# B&R Automation Studio project vibratorControlWithCurrentController (part 18)

#### simWing.st
```iecst
ACTION simWing:

	IF wing.activated THEN

		//===============================================================================
		//						Read outputs
		//===============================================================================
		//upperOpen
		wing.hw.out[0].enable := TRUE;
		wing.hw.out[0].pvName := 'upperFlap:this.hw.do_open';
		wing.hw.out[0]();

		//middleOpen
		wing.hw.out[1].enable := TRUE;
		wing.hw.out[1].pvName := 'middleFlap:this.hw.do_open';
		wing.hw.out[1]();

		//bottomOpen
		wing.hw.out[2].enable := TRUE;
		wing.hw.out[2].pvName := 'bottomFlap:this.hw.do_open';
		wing.hw.out[2]();

		//===============================================================================
		//						Set inputs
		//===============================================================================
		//::upperFlap:this.flap.di_changeover
		wing.hw.in[0].enable   := TRUE;
		wing.hw.in[0].dpName   := '%IX.IF6.ST5.DigitalInput01';

		//::middleFlap:this.flap.di_changeover
		wing.hw.in[1].enable   := TRUE;
		wing.hw.in[1].dpName   := '%IX.IF6.ST5.DigitalInput03';

		//::bottomFlap:this.flap.di_changeover
		wing.hw.in[2].enable   := TRUE;
		wing.hw.in[2].dpName   := '%IX.IF6.ST5.DigitalInput02';

		FOR i:=0 TO MAX_WINGS DO
			wing.var.TON_delay[i].PT := T#50ms;
			wing.var.TOF_changeOver[i].PT := T#20ms;
			// check for change
			IF wing.var.oldVal[i] <> wing.hw.out[i].actValue THEN
				wing.var.TON_delay[i].IN := TRUE;
			END_IF
			// after delay time
			wing.var.TOF_changeOver[i].IN := wing.var.TON_delay[i].Q;

			IF wing.var.TOF_changeOver[i].Q THEN
				wing.var.TON_delay[i].IN := FALSE;
				wing.hw.in[i].setValue := 1;
			ELSE
				wing.hw.in[i].setValue := 0;
			END_IF

			wing.var.TON_delay[i]();
			wing.var.TOF_changeOver[i]();
			wing.var.oldVal[i] := wing.hw.out[i].actValue;
		END_FOR

		wing.hw.in[0]();
		wing.hw.in[1]();
		wing.hw.in[2]();

	END_IF

	IF gWingInterface.status.simNeighbour OR wing.activated THEN
		//neighbourBottomOpen
		wing.hw.out[3].enable := TRUE;
		wing.hw.out[3].pvName := 'bottomFlap:this.hw.do_neighbourOpen';
		wing.hw.out[3]();

		//bricksInMiddle
		wing.hw.out[4].enable := TRUE;
		wing.hw.out[4].pvName := 'cassette:this.hw.do_bricksReadyInCassette';
		wing.hw.out[4]();

		//bricksInMiddle
		wing.hw.out[5].enable := TRUE;
		wing.hw.out[5].pvName := 'bottomFlap:this.hw.do_neighbourPortionReady';
		wing.hw.out[5]();

		//::bottomFlap:this.neighbourFlap.di_changeover
		wing.hw.in[3].enable   := TRUE;
		wing.hw.in[3].dpName   := '%IX.IF6.ST5.DigitalInput04';

		 i:=3;
		wing.var.TON_delay[i].PT := T#50ms;
		wing.var.TOF_changeOver[i].PT := T#20ms;
		// check for change
		IF wing.var.oldVal[i] <> wing.hw.out[i].actValue THEN
			wing.var.TON_delay[i].IN := TRUE;
		END_IF
		// after delay time
		wing.var.TOF_changeOver[i].IN := wing.var.TON_delay[i].Q;

		IF wing.var.TOF_changeOver[i].Q THEN
			wing.var.TON_delay[i].IN := FALSE;
			wing.hw.in[i].setValue := 1;
		ELSE
			wing.hw.in[i].setValue := 0;
		END_IF

		wing.var.TON_delay[i]();
		wing.var.TOF_changeOver[i]();
		wing.var.oldVal[i] := wing.hw.out[i].actValue;

		wing.hw.in[3]();

		//::bottomFlap:this.hw.di_neighbourActive
		wing.hw.in[4].enable   := gWingInterface.status.simNeighbour;
		wing.hw.in[4].dpName   := '%IX.IF6.ST6.DigitalInput02';
		wing.hw.in[4].setValue := 1;
		wing.hw.in[4]();

		//::bottomFlap:this.hw.di_neighbourPortionReady
		wing.hw.in[5].enable   :=  gWingInterface.status.simNeighbour;
		wing.hw.in[5].dpName   := '%IX.IF6.ST6.DigitalInput05';
		IF wing.hw.out[5].actValue > 0 THEN
			wing.hw.in[5].setValue := 1;
		ELSE
			wing.hw.in[5].setValue := 0;
		END_IF
		wing.hw.in[5]();

	END_IF

END_ACTION
```

#### simCassette.st
```iecst
ACTION simCassette:

	IF cassette.activated THEN
		gCassetteInterface.cmd.cassetteIsBeingSimulated := TRUE;
		// init sim (TRUE = no box)
		IF EDGEPOS(cassette.activated) THEN
			cassette.hw.in[0].setValue := TRUE;
			cassette.hw.in[1].setValue := TRUE;
		END_IF

		//===============================================================================
		//						Read outputs
		//===============================================================================
		//cassette:this.hw.do_bricksReadyInCassette
		cassette.hw.out[0].enable := TRUE;
		cassette.hw.out[0].pvName := 'cassette:this.hw.do_bricksReadyInCassette';
		cassette.hw.out[0]();

		//cassette:this.hw.do_cassetteRelease
		cassette.hw.out[1].enable := TRUE;
		cassette.hw.out[1].pvName := 'cassette:this.hw.do_cassetteRelease';
		cassette.hw.out[1]();

		//===============================================================================
		//						Set inputs
		//===============================================================================

		cassette.hw.in[0].enable   := TRUE;
		cassette.hw.in[0].dpName   := '%IX.IF6.ST6.DigitalInput03';		//cassette:this.hw.di_cassetteReady

		cassette.hw.in[1].enable   := TRUE;
		cassette.hw.in[1].dpName   := '%IX.IF6.ST6.DigitalInput01';		//cassette:this.hw.di_cassetteQueue

		//cassette:this.hw.di_cassetteQueue
		CASE cassette.var.state OF
			0:
				cassette.hw.in[0].setValue := 0; // no cassette on ready sensor

				cassette.var.tonDelay(IN := TRUE, PT:=cassette.var.toReadyTime);

				IF cassette.var.tonDelay.Q THEN
					cassette.var.tonDelay(IN:=FALSE);
					cassette.var.state := 10;
				END_IF
			10:
				cassette.var.tonDelay(IN := cassette.hw.out[1].actValue > 0, PT:=cassette.var.toReadyTime);

				IF cassette.var.tonDelay.Q THEN
					cassette.var.tonDelay(IN:=FALSE);
					cassette.var.state := 20;
				END_IF

			20:
				cassette.hw.in[0].setValue := 1; // cassette on ready sensor

				cassette.var.tonDelay(IN := TRUE, PT:=cassette.var.fromReadyTime);

				IF cassette.var.tonDelay.Q THEN
					cassette.var.tonDelay(IN:=FALSE);
					cassette.var.tofDelay(IN := TRUE, PT:=cassette.var.cassetteQueueTime);
					cassette.var.state := 0;
				END_IF
		END_CASE

		cassette.var.tofDelay(IN := FALSE, PT:=cassette.var.toReadyTime);
		cassette.hw.in[1].setValue := SEL(cassette.var.tofDelay.Q, 1, 0); // no cassette on queue sensor

	cassette.hw.in[0]();
	cassette.hw.in[1]();

	IF gWingInterface.status.simNeighbour THEN
		//cassette:this.hw.di_neighbourBricksInCassette
		cassette.hw.in[2].enable   := TRUE;
			cassette.hw.in[2].dpName   := '%IX.IF6.ST6.DigitalInput07';
			IF cassette.hw.out[0].actValue > 0 THEN // this machine has brics ready then wing do also.
				cassette.hw.in[2].setValue := 1;
			ELSE
				cassette.hw.in[2].setValue := 0;
			END_IF
		ELSE
			cassette.hw.in[2].enable   := FALSE;
		END_IF
		cassette.hw.in[2]();

	ELSE
		gCassetteInterface.cmd.cassetteIsBeingSimulated := FALSE;
	END_IF

END_ACTION
```

### simGlobal.typ
```iecst
TYPE
	gSimulation_status_typ : 	STRUCT
		photoSensor : BOOL;
		simulateAllButWing : BOOL;
	END_STRUCT;
	gSimulation_typ : 	STRUCT
		status : gSimulation_status_typ;
	END_STRUCT;
END_TYPE
```

### simGlobal.var
```iecst
VAR
	gSimulation : gSimulation_typ;
END_VAR
```

### simCapconGlobal.typ - Global data types
```iecst
TYPE
	gSimCapcon_typ : 	STRUCT
		cmd : gSimCapcon_cmd_typ; (*Command type.*)
		status : gSimCapcon_status_typ; (*Status type.*)
		parameter : gSimCapcon_parameter_typ;
	END_STRUCT;
	gSimCapcon_cmd_typ : 	STRUCT  (*Global command type.*)
		readFile : BOOL;
	END_STRUCT;
	gSimCapcon_status_typ : 	STRUCT  (*Global status type.*)
		data : gSimCapcon_data_typ;
		simSignal : INT;
	END_STRUCT;
	gSimCapcon_parameter_typ : 	STRUCT
		fileName : STRING[200];
	END_STRUCT;
	gSimCapcon_data_typ : 	STRUCT
		record : ARRAY[0..CAPCON_LOG_RECORD_SIZE]OF gSimCapcon_data_record_typ;
	END_STRUCT;
	gSimCapcon_data_record_typ : 	STRUCT
		value : ARRAY[0..CAPCON_LOG_SAMPLE_SIZE]OF INT;
	END_STRUCT;
END_TYPE
```

### simCapconGlobal.var - Global variables
```iecst
VAR
	gSimCapcon : gSimCapcon_typ; (*Global recipe interface.*)
END_VAR
VAR CONSTANT
	CAPCON_LOG_RECORD_SIZE : DINT := 99; (*99 means 100*)
	CAPCON_LOG_SAMPLE_SIZE : DINT := 499; (*499 means 500*)
END_VAR
```

### Program Logical/simulation/capcon/simCapcon (IEC)

#### main.st - Init, cyclic, exit code
```iecst
PROGRAM _INIT

	gSimCapcon.parameter.fileName := 'simData.csv';

	IF gMainInterface.status.simulation THEN
		gSimCapcon.cmd.readFile := TRUE;
	END_IF

END_PROGRAM

PROGRAM _CYCLIC

	CASE cm.state OF

		0:
			cm.description := 'waiting for command';
			IF gSimCapcon.cmd.readFile THEN
				gSimCapcon.cmd.readFile := FALSE;
				cm.state := 100;
			END_IF

		10:

		100:
			cm.description := 'wait for open file ok';
			this.FileOpen_0.enable 	:= TRUE;
			this.FileOpen_0.pDevice := ADR('SIMDATA');
			this.FileOpen_0.pFile 	:= ADR(gSimCapcon.parameter.fileName);
			this.FileOpen_0.mode 	:= fiREAD_ONLY;
			this.FileOpen_0();
			IF this.FileOpen_0.status = ERR_OK THEN
				brdkStrMemSet(ADR(this.tmpData),0,SIZEOF(this.tmpData));
				this.FileRead_0.ident 	:= this.FileOpen_0.ident;
				this.FileRead_0.offset 	:= 0;
				this.FileRead_0.pDest 	:= ADR(this.tmpData);
				this.FileRead_0.len 	:= SIZEOF(this.tmpData);
				this.FileRead_0.enable	:= TRUE;
				cm.state 				:= 110;
			END_IF

		110:
			cm.description := 'waiting for read file';
			this.FileRead_0();
			IF this.FileRead_0.status = ERR_OK THEN
				this.FileRead_0(enable := FALSE);
				this.FileClose_0.enable := TRUE;
				this.FileClose_0.ident 	:= this.FileOpen_0.ident;
				cm.state := 120;
			END_IF

		120:
			cm.description := 'waiting for file close';
			this.FileClose_0();
			IF this.FileClose_0.status = ERR_OK THEN
				this.FileOpen_0(enable := FALSE);
				this.FileClose_0(enable := FALSE);
				this.lfCnt := 0;
				this.offset := 0;
				brdkStrMemSet(ADR(this.tmpStr),0,SIZEOF(this.tmpStr));
				cm.state := 130;
			END_IF

		130:
			cm.description := 'parse a line';
			FOR this.offset := this.offset TO MAX_FILE_SIZE DO
				CASE this.tmpData[this.offset] OF

					0:	// found end of file
						cm.state := 0;
						EXIT;

					10: // found a line feed
						this.lfCnt 		:= this.lfCnt + 1;
						this.colCnt 	:= 0;					// reset ; count

					59:	// found a ;
						IF this.lfCnt >= START_LINE_FEEDS AND this.colCnt >= START_COLS AND this.colCnt <= MAX_COLS THEN
							gSimCapcon.status.data.record[this.lfCnt - START_LINE_FEEDS].value[this.colCnt - START_COLS] := DINT_TO_INT(brdkStrAToDint(ADR(this.tmpStr),BRDK_STR_CONVERT_DECIMAL));
							brdkStrMemSet(ADR(this.tmpStr),0,SIZEOF(this.tmpStr));
							this.charCnt := 0;
						END_IF
						this.colCnt := this.colCnt + 1;

					32..57:	// numbers and some signs
						IF this.lfCnt >= START_LINE_FEEDS AND this.colCnt >= START_COLS AND this.colCnt <= MAX_COLS THEN
							this.tmpStr[this.charCnt] := this.tmpData[this.offset];
							this.charCnt := this.charCnt + 1;
						END_IF

				END_CASE

			END_FOR

	END_CASE

	cm;

END_PROGRAM

PROGRAM _EXIT
	(* Insert code here *)

END_PROGRAM
```

#### types.typ - Local data types
```iecst
TYPE
	local_typ : 	STRUCT
		FileOpen_0 : FileOpen;
		FileRead_0 : FileRead;
		FileClose_0 : FileClose;
		tmpData : ARRAY[0..MAX_FILE_SIZE]OF USINT;
		offset : UDINT;
		tmpStr : ARRAY[0..9]OF USINT;
		colCnt : UINT;
		lfCnt : USINT;
		charCnt : USINT;
	END_STRUCT;
END_TYPE
```

#### variables.var - Local variables
```iecst
VAR
	this : local_typ;
END_VAR
VAR CONSTANT
	MAX_FILE_SIZE : UDINT := 1000000;
END_VAR
VAR
	cm : brdkCM;
END_VAR
VAR CONSTANT
	MAX_COLS : UINT := 499; (*maximum number of ;*)
	START_COLS : UINT := 2; (*number of ; in a line before the data is good*)
	START_LINE_FEEDS : USINT := 5; (*number of line feeds before the data is good*)
END_VAR
```

### Data object Logical/gAxisVibCobj/gAxisVibCi (Ax)

#### gAxisVibCi.ax
```
InitParameter (Version=5.23.1, NcSwId=ACP10)
  ACP10AXIS_typ:
    dig_in:
      level:
        reference = ncACTIV_HI
        pos_hw_end = ncACTIV_HI
        neg_hw_end = ncACTIV_HI
        trigger1 = ncACTIV_HI
        trigger2 = ncACTIV_HI
    encoder_if:
      parameter:
        count_dir = ncSTANDARD
        scaling:
          load:
            units = 1000
            rev_motor = 1
    limit:
      parameter:
        v_pos = 54000.0
        v_neg = 54000.0
        a1_pos = 5000000.0
        a2_pos = 5000000.0
        a1_neg = 5000000.0
        a2_neg = 5000000.0
        t_jolt = 0.0
        t_in_pos = 0.0
        pos_sw_end = 8388607
        neg_sw_end = -8388608
        ds_warning = 500.0
        ds_stop = 1000.0
        a_stop = 1.0E+30
        dv_stop = 0.0
        dv_stop_mode = ncOFF
    controller:
      mode = ncUF
      position:
        kv = 50.0
        tn = 0.0
        t_predict = 0.0004
        t_total = 0.0004
        p_max = 1.0E+30
        i_max = 0.0
      speed:
        kv = 2.0
        tn = 0.0
        t_filter = 0.0
        isq_filter1:
          type = ncOFF
          a0 = 0.0
          a1 = 0.0
          b0 = 0.0
          b1 = 0.0
          b2 = 0.0
          c0_par_id = 0
          c1_par_id = 0
        isq_filter2:
          type = ncOFF
          a0 = 0.0
          a1 = 0.0
          b0 = 0.0
          b1 = 0.0
          b2 = 0.0
          c0_par_id = 0
          c1_par_id = 0
        isq_filter3:
          type = ncOFF
          a0 = 0.0
          a1 = 0.0
          b0 = 0.0
          b1 = 0.0
          b2 = 0.0
          c0_par_id = 0
          c1_par_id = 0
      uf:
        type = ncLINEAR
        auto_config = ncOFF
        u0 = 0.0
        un = 0.0
        fn = 50.0
        k_f_slip = 0.0
      ff:
        mode = ncSTANDARD
        torque_load = 0.0
        torque_pos = 0.0
        torque_neg = 0.0
        kv_torque = 0.0
        inertia = 0.0
        t_filter_a = 0.0
      fb:
        mode = ncSTANDARD
        speed_mix_ratio = 0.0
        speed_kv = 2.0
      model:
        mass1:
          inertia = 0.0
          viscous_friction = 0.0
        mass2:
          inertia = 0.0
          viscous_friction = 0.0
          stiffness = 0.0
          damping = 0.0
    move:
      stop:
        parameter[0]:
          decel_ramp = ncA_LIMIT
          controller = ncON
        parameter[1]:
          decel_ramp = ncA_LIMIT
          controller = ncON
        parameter[2]:
          decel_ramp = ncA_LIMIT
          controller = ncON
        parameter[3]:
          decel_ramp = ncA_LIMIT
          controller = ncON
        quickstop:
          decel_ramp = ncA_LIMIT
          t_jolt = 0.0
        drive_error:
          decel_ramp = ncA_LIMIT
      homing:
        parameter:
          s = 0
          v_switch = 5000.0
          v_trigger = 500.0
          a = 50000.0
          mode = ncDIRECT
          edge_sw = ncPOSITIVE
          start_dir = ncPOSITIVE
          trigg_dir = ncPOSITIVE
          ref_pulse = ncOFF
          fix_dir = ncOFF
          tr_s_block = 0.0
          torque_lim = 0.0
          ds_block = 0.0
          ds_stop = 0.0
      basis:
        parameter:
          v_pos = 50000.0
          v_neg = 50000.0
          a1_pos = 500000.0
          a2_pos = 500000.0
          a1_neg = 500000.0
          a2_neg = 500000.0
    message:
      text:
        parameter:
          format = ncZERO
          columns = 81
          data_modul = acp10etxen
```

### Data object Logical/gAxisVibCobj/cfCurCtr (Apt)

#### cfCurCtr.apt
```
AcoposParameterTable:
  Root Parameters:
    128 = 1 (Name=SGEN_SW_END_IGNORE)  // Limit values: Ignore SW end positions
    652 = 0 (Name=MOTOR_ENCOD_ATTR)  // Motor: Encoder: Attribute
    1215 = 0 (Name=MOTOR_TEMPSENS_TYPE)  // Temperature sensor: Type
    90 = 76 (Name=BRAKE_MODE)  // Motor holding brake: Mode
    1208 = 1 (Name=MOTOR_NUM_PHASES)  // Motor: Number of motor phases
    Axis Parameter Identification, Synchronous Motor:
      Group  // General Parameters
        30 = 2 (Name=MOTOR_TYPE)  // Motor: Type
        31 = 0x0203 (Name=MOTOR_COMPATIBILITY)  // Motor: Software compatibility
        46 = 1 (Name=MOTOR_WIND_CONNECT)  // Motor: Winding connection
        62 = 0 (Name=MOTOR_INERTIA, Unit=kgm²)  // Motor: Moment of inertia
        849 = 0 (Name=MOTOR_TAU_THERM, Unit=s)  // Motor: Thermal time constant
      Group  // Brake Parameters
        42 = 0 (Name=MOTOR_BRAKE_CURR_RATED, Unit=A)  // Motor holding brake: Rated current
        43 = 0 (Name=MOTOR_BRAKE_TORQ_RATED, Unit=Nm)  // Motor holding brake: Rated torque
        44 = 0 (Name=MOTOR_BRAKE_ON_TIME, Unit=s)  // Motor holding brake: Engaging delay
        45 = 0 (Name=MOTOR_BRAKE_OFF_TIME, Unit=s)  // Motor holding brake: Release delay
      Group  // Thermo Sensor Parameters
        64 = 0 (Name=MOTOR_TEMPSENS_PAR1)  // Temperature sensor: Parameter 1
        65 = 0 (Name=MOTOR_TEMPSENS_PAR2)  // Temperature sensor: Parameter 2
        66 = 0 (Name=MOTOR_TEMPSENS_PAR3)  // Temperature sensor: Parameter 3
        67 = 0 (Name=MOTOR_TEMPSENS_PAR4)  // Temperature sensor: Parameter 4
        68 = 0 (Name=MOTOR_TEMPSENS_PAR5)  // Temperature sensor: Parameter 5
        69 = 0 (Name=MOTOR_TEMPSENS_PAR6)  // Temperature sensor: Parameter 6
        70 = 0 (Name=MOTOR_TEMPSENS_PAR7)  // Temperature sensor: Parameter 7
        71 = 0 (Name=MOTOR_TEMPSENS_PAR8)  // Temperature sensor: Parameter 8
        72 = 0 (Name=MOTOR_TEMPSENS_PAR9)  // Temperature sensor: Parameter 9
        73 = 0 (Name=MOTOR_TEMPSENS_PAR10)  // Temperature sensor: Parameter 10
        74 = 50 (Name=MOTOR_WIND_TEMP_MAX, Unit=°C)  // Temperature sensor: Limit temperature
      Group  // Result Parameters of Parameter Identification
        47 = 1 (Name=MOTOR_POLEPAIRS)  // Motor: Number of pole-pairs
        48 = 200 (Name=MOTOR_VOLTAGE_RATED, Unit=V)  // Motor: Rated voltage
        50 = 6000 (Name=MOTOR_SPEED_RATED, Unit=1/min)  // Motor: Rated speed
        51 = 6600 (Name=MOTOR_SPEED_MAX, Unit=1/min)  // Motor: Maximum speed
        52 = 1 (Name=MOTOR_TORQ_STALL, Unit=Nm)  // Motor: Stall torque
        53 = 1 (Name=MOTOR_TORQ_RATED, Unit=Nm)  // Motor: Rated torque
        54 = 1 (Name=MOTOR_TORQ_MAX, Unit=Nm)  // Motor: Peak torque
        56 = 1 (Name=MOTOR_CURR_STALL, Unit=A)  // Motor: Stall current
        58 = 4 (Name=MOTOR_CURR_MAX, Unit=A)  // Motor: Peak current
        57 = 3.77 (Name=MOTOR_CURR_RATED, Unit=A)  // Motor: Rated current
        59 = 1 (Name=MOTOR_WIND_CROSS_SECT, Unit=mm²)  // Motor: Line cross section
        60 = 6.917 (Name=MOTOR_STATOR_RESISTANCE, Unit=Ohm)  // Motor: Stator resistance
        61 = 0.3237 (Name=MOTOR_STATOR_INDUCTANCE, Unit=Henry)  // Motor: Stator inductance
        1208 = 1 (Name=MOTOR_NUM_PHASES)  // Motor: Number of motor phases
      IPL:
        777 = IPL_MODE+0 (Name=FUNCTION_BLOCK_CREATE, Disabled=FALSE)  // Function block: Create a FB instance
        8712 = USER_R4_VAR1 (Name=IPL_IN_PARID+0, Disabled=FALSE)  // FB0 FB IPL: Parameter ID of input
        8760 = CYCLIC_TODRV_COUNT (Name=IPL_EV_PARID+0)  // FB0 FB IPL: Parameter ID of event input
        8720 = 800 (Name=IPL_CYCLE_TIME+0, Unit=us)  // FB0 FB IPL: Cycle time
        8704 = 2 (Name=IPL_MODE+0, Disabled=FALSE)  // FB0 FB IPL: Mode - (4) quadric no overshoot
      Group:
        347 = 10000 (Name=F_SWITCH, Unit=cps)  // Inverter: Switch frequency
        49 = 100 (Name=MOTOR_VOLTAGE_CONST, Unit=mV*min)  // Motor: Voltage constant
        813 = 0  // PARID_SIGEN_OFFS
        55 = 3 (Name=MOTOR_TORQ_CONST, Unit=Nm/A)  // Motor: Torque constant
        63 = 0 (Name=MOTOR_COMMUT_OFFSET, Unit=rad)  // Motor: Commutation offset
        713 = 8752 (Name=ICTRL_SET_PARID)  // CTRL Current controller: Set value parameter ID of stator current quadrature component
        1480 = 0 (Name=TLIM_MODE)  // CTRL Torque limiter: Mode
        1569 = 2500 (Name=ICTRL_US_FILTER1_A0)  // CTRL Current: Set voltage filter coefficient A0
        1570 = 2200 (Name=ICTRL_US_FILTER1_A1)  // CTRL Current: Set voltage filter coefficient A1
        1568 = 1 (Name=ICTRL_US_FILTER_TYPE)  // CTRL Current: Set voltage filter type
        1166 = 0 (Name=ICTRL_AUTO_CONFIG)  // CTRL Current: Automatic configuration
        223 = 300 (Name=ICTRL_KV, Unit=V/A)  // CTRL Current controller: Proportional amplification factor
        225 = 0.00526 (Name=ICTRL_TI, Unit=s)  // CTRL Current controller: Integral action time
        328 = 5 (Name=CONTROLLER_MODE)  // CTRL Controller: Mode
      Voltage observer:
        1354 = 1 (Name=OBS_MODE_BITS)  // Observer: Mode bits
        1298 = 25.4481 (Name=OBS_VOLT_INVCL_A1)  // Voltage observer: Inverter adjustment amplification factor
        1299 = 2.2113 (Name=OBS_VOLT_INVCL_A2, Unit=1/A)  // Voltage observer: Inverter adjustment exponent
    232 = 0 (Name=CYCLIC_TODRV_PAR_INDEX)  // Cyclic communication: Parameter index of data to drive
    207 = CYCLIC_FRDRV_REC_INDEX (Name=CYCLIC_TODRV_PARID)  // Cyclic communication: Parameter ID of data to drive
    777 = ARITH_MODE+0 (Name=FUNCTION_BLOCK_CREATE)  // Function block: Create a FB instance
    777 = DYNSYS_MODE+0 (Name=FUNCTION_BLOCK_CREATE)  // Function block: Create a FB instance
    777 = ARITH_MODE+1 (Name=FUNCTION_BLOCK_CREATE)  // Function block: Create a FB instance
    777 = ARITH_MODE+2 (Name=FUNCTION_BLOCK_CREATE)  // Function block: Create a FB instance
    777 = DYNSYS_MODE+1 (Name=FUNCTION_BLOCK_CREATE)  // Function block: Create a FB instance
    777 = DYNSYS_MODE+2 (Name=FUNCTION_BLOCK_CREATE)  // Function block: Create a FB instance
    777 = DYNSYS_MODE+3 (Name=FUNCTION_BLOCK_CREATE)  // Function block: Create a FB instance
    777 = DYNSYS_MODE+4 (Name=FUNCTION_BLOCK_CREATE)  // Function block: Create a FB instance
    777 = VAR_I4_0+0 (Name=FUNCTION_BLOCK_CREATE)  // Function block: Create a FB instance
    777 = VAR_R4_0+0 (Name=FUNCTION_BLOCK_CREATE)  // Function block: Create a FB instance
    777 = MINMAX_MODE+0 (Name=FUNCTION_BLOCK_CREATE)  // Function block: Create a FB instance
    777 = MINMAX_MODE+1 (Name=FUNCTION_BLOCK_CREATE)  // Function block: Create a FB instance
    777 = COUNT_MODE+0 (Name=FUNCTION_BLOCK_CREATE)  // Function block: Create a FB instance
    777 = FILTER_MODE+0 (Name=FUNCTION_BLOCK_CREATE)  // Function block: Create a FB instance
    ARITH EMF:
      3584 = 0 (Name=ARITH_MODE+0)  // FB0 ARITH Mode
      3592 = 216 (Name=ARITH_IN1_PARID+0)  // FB0 ARITH Parameter ID of input1
      3600 = 214 (Name=ARITH_IN2_PARID+0)  // FB0 ARITH Parameter ID of input2
      3632 = 1 (Name=ARITH_K1+0)  // FB0 ARITH Multiplication factor1
      3640 = -4.2 (Name=ARITH_K2+0)  // FB0 ARITH Multiplication factor2
      3584 = 4 (Name=ARITH_MODE+0)  // FB0 ARITH Mode
    DYNSYS Integrate EMF:
      14336 = 0 (Name=DYNSYS_MODE+0)  // FB0 FB DYNSYS: Mode
      14344 = 0.99 (Name=DYNSYS_PAR_A+0)  // FB0 FB DYNSYS: System parameter A
      14344 = 0.0002 (Name=DYNSYS_PAR_A+0)  // FB0 FB DYNSYS: System parameter A
      14344 = 0 (Name=DYNSYS_PAR_A+0)  // FB0 FB DYNSYS: System parameter A
      14344 = 0 (Name=DYNSYS_PAR_A+0)  // FB0 FB DYNSYS: System parameter A
      14344 = 0 (Name=DYNSYS_PAR_A+0)  // FB0 FB DYNSYS: System parameter A
      14344 = 0 (Name=DYNSYS_PAR_A+0)  // FB0 FB DYNSYS: System parameter A
      14344 = 0 (Name=DYNSYS_PAR_A+0)  // FB0 FB DYNSYS: System parameter A
      14344 = 0 (Name=DYNSYS_PAR_A+0)  // FB0 FB DYNSYS: System parameter A
      14344 = 0 (Name=DYNSYS_PAR_A+0)  // FB0 FB DYNSYS: System parameter A
      14352 = 0.0002 (Name=DYNSYS_PAR_B+0)  // FB0 FB DYNSYS: System parameter B
      14352 = 0 (Name=DYNSYS_PAR_B+0)  // FB0 FB DYNSYS: System parameter B
      14352 = 1 (Name=DYNSYS_PAR_B+0)  // FB0 FB DYNSYS: System parameter B
      14352 = 0 (Name=DYNSYS_PAR_B+0)  // FB0 FB DYNSYS: System parameter B
      14352 = 0 (Name=DYNSYS_PAR_B+0)  // FB0 FB DYNSYS: System parameter B
      14352 = 1 (Name=DYNSYS_PAR_B+0)  // FB0 FB DYNSYS: System parameter B
      14360 = 1 (Name=DYNSYS_PAR_C+0)  // FB0 FB DYNSYS: System parameter C
      14360 = 0 (Name=DYNSYS_PAR_C+0)  // FB0 FB DYNSYS: System parameter C
      14360 = 0 (Name=DYNSYS_PAR_C+0)  // FB0 FB DYNSYS: System parameter C
      14360 = 0 (Name=DYNSYS_PAR_C+0)  // FB0 FB DYNSYS: System parameter C
      14360 = 0 (Name=DYNSYS_PAR_C+0)  // FB0 FB DYNSYS: System parameter C
      14360 = 1 (Name=DYNSYS_PAR_C+0)  // FB0 FB DYNSYS: System parameter C
      14408 = ARITH_VALUE_R4+0 (Name=DYNSYS_IN1_PARID+0)  // FB0 FB DYNSYS: Parameter ID for input 1
      14416 = 214 (Name=DYNSYS_IN2_PARID+0)  // FB0 FB DYNSYS: Parameter ID for input 2
      14336 = 1 (Name=DYNSYS_MODE+0)  // FB0 FB DYNSYS: Mode (note: set SCTRL_ADD_SET_PARID = DYNSYS_OUT1_VALUE+X for activation)
    ARITH Airgap:
      3585 = 0 (Name=ARITH_MODE+1)  // FB0 ARITH Mode
      3593 = DYNSYS_OUT2_VALUE+0 (Name=ARITH_IN1_PARID+1)  // FB0 ARITH Parameter ID of input1
      3601 = DYNSYS_OUT1_VALUE+0 (Name=ARITH_IN2_PARID+1)  // FB0 ARITH Parameter ID of input2
      3585 = 5 (Name=ARITH_MODE+1)  // FB0 ARITH Mode
    ARITH Observer:
      3586 = 0 (Name=ARITH_MODE+2)  // FB2 FB ARITH: Mode
      3594 = 1296 (Name=ARITH_IN1_PARID+2)  // FB2 FB ARITH: Parameter ID of input1
      3602 = 1297 (Name=ARITH_IN2_PARID+2)  // FB2 FB ARITH: Parameter ID of input2
      3586 = 2 (Name=ARITH_MODE+2)  // FB2 FB ARITH: Mode
    DYNSYS+1:
      14337 = 0 (Name=DYNSYS_MODE+1)  // FB0 FB DYNSYS: Mode
      14345 = 0 (Name=DYNSYS_PAR_A+1)  // FB0 FB DYNSYS: System parameter A
      14345 = 0 (Name=DYNSYS_PAR_A+1)  // FB0 FB DYNSYS: System parameter A
      14345 = 0 (Name=DYNSYS_PAR_A+1)  // FB0 FB DYNSYS: System parameter A
      14345 = 0 (Name=DYNSYS_PAR_A+1)  // FB0 FB DYNSYS: System parameter A
      14345 = 1 (Name=DYNSYS_PAR_A+1)  // FB0 FB DYNSYS: System parameter A
      14345 = 0 (Name=DYNSYS_PAR_A+1)  // FB0 FB DYNSYS: System parameter A
      14345 = 0 (Name=DYNSYS_PAR_A+1)  // FB0 FB DYNSYS: System parameter A
      14345 = 0 (Name=DYNSYS_PAR_A+1)  // FB0 FB DYNSYS: System parameter A
      14345 = 0 (Name=DYNSYS_PAR_A+1)  // FB0 FB DYNSYS: System parameter A
      14345 = 1 (Name=DYNSYS_PAR_A+1)  // FB0 FB DYNSYS: System parameter A
      14345 = 0 (Name=DYNSYS_PAR_A+1)  // FB0 FB DYNSYS: System parameter A
      14345 = 0 (Name=DYNSYS_PAR_A+1)  // FB0 FB DYNSYS: System parameter A
      14345 = 0 (Name=DYNSYS_PAR_A+1)  // FB0 FB DYNSYS: System parameter A
      14345 = 0 (Name=DYNSYS_PAR_A+1)  // FB0 FB DYNSYS: System parameter A
      14345 = 1 (Name=DYNSYS_PAR_A+1)  // FB0 FB DYNSYS: System parameter A
      14345 = 0 (Name=DYNSYS_PAR_A+1)  // FB0 FB DYNSYS: System parameter A
      14353 = 1 (Name=DYNSYS_PAR_B+1)  // FB1 FB DYNSYS: System parameter B
      14353 = 0 (Name=DYNSYS_PAR_B+1)  // FB1 FB DYNSYS: System parameter B
      14353 = 0 (Name=DYNSYS_PAR_B+1)  // FB1 FB DYNSYS: System parameter B
      14353 = 0 (Name=DYNSYS_PAR_B+1)  // FB1 FB DYNSYS: System parameter B
      14361 = 1 (Name=DYNSYS_PAR_C+1)  // FB1 FB DYNSYS: System parameter C
      14361 = 0 (Name=DYNSYS_PAR_C+1)  // FB1 FB DYNSYS: System parameter C
      14361 = 0 (Name=DYNSYS_PAR_C+1)  // FB1 FB DYNSYS: System parameter C
      14361 = 0 (Name=DYNSYS_PAR_C+1)  // FB1 FB DYNSYS: System parameter C
      14361 = 0 (Name=DYNSYS_PAR_C+1)  // FB1 FB DYNSYS: System parameter C
      14361 = 1 (Name=DYNSYS_PAR_C+1)  // FB1 FB DYNSYS: System parameter C
      14361 = 0 (Name=DYNSYS_PAR_C+1)  // FB1 FB DYNSYS: System parameter C
      14361 = 0 (Name=DYNSYS_PAR_C+1)  // FB1 FB DYNSYS: System parameter C
      14409 = 216 (Name=DYNSYS_IN1_PARID+1)  // FB0 FB DYNSYS: Parameter ID for input 1
      14337 = 1 (Name=DYNSYS_MODE+1)  // FB0 FB DYNSYS: Mode (note: set SCTRL_ADD_SET_PARID = DYNSYS_OUT1_VALUE+X for activation)
    DYNSYS+2:
      14338 = 0 (Name=DYNSYS_MODE+2)  // FB0 FB DYNSYS: Mode
      14346 = 0 (Name=DYNSYS_PAR_A+2)  // FB0 FB DYNSYS: System parameter A
      14346 = 0 (Name=DYNSYS_PAR_A+2)  // FB0 FB DYNSYS: System parameter A
      14346 = 0 (Name=DYNSYS_PAR_A+2)  // FB0 FB DYNSYS: System parameter A
      14346 = 0 (Name=DYNSYS_PAR_A+2)  // FB0 FB DYNSYS: System parameter A
      14346 = 1 (Name=DYNSYS_PAR_A+2)  // FB0 FB DYNSYS: System parameter A
      14346 = 0 (Name=DYNSYS_PAR_A+2)  // FB0 FB DYNSYS: System parameter A
      14346 = 0 (Name=DYNSYS_PAR_A+2)  // FB0 FB DYNSYS: System parameter A
      14346 = 0 (Name=DYNSYS_PAR_A+2)  // FB0 FB DYNSYS: System parameter A
      14346 = 0 (Name=DYNSYS_PAR_A+2)  // FB0 FB DYNSYS: System parameter A
      14346 = 1 (Name=DYNSYS_PAR_A+2)  // FB0 FB DYNSYS: System parameter A
      14346 = 0 (Name=DYNSYS_PAR_A+2)  // FB0 FB DYNSYS: System parameter A
      14346 = 0 (Name=DYNSYS_PAR_A+2)  // FB0 FB DYNSYS: System parameter A
      14346 = 0 (Name=DYNSYS_PAR_A+2)  // FB0 FB DYNSYS: System parameter A
      14346 = 0 (Name=DYNSYS_PAR_A+2)  // FB0 FB DYNSYS: System parameter A
      14346 = 1 (Name=DYNSYS_PAR_A+2)  // FB0 FB DYNSYS: System parameter A
      14346 = 0 (Name=DYNSYS_PAR_A+2)  // FB0 FB DYNSYS: System parameter A
      14354 = 1 (Name=DYNSYS_PAR_B+2)  // FB2 FB DYNSYS: System parameter B
      14354 = 0 (Name=DYNSYS_PAR_B+2)  // FB2 FB DYNSYS: System parameter B
      14354 = 0 (Name=DYNSYS_PAR_B+2)  // FB2 FB DYNSYS: System parameter B
      14354 = 0 (Name=DYNSYS_PAR_B+2)  // FB2 FB DYNSYS: System parameter B
      14362 = 0 (Name=DYNSYS_PAR_C+2)  // FB2 FB DYNSYS: System parameter C
      14362 = 0 (Name=DYNSYS_PAR_C+2)  // FB2 FB DYNSYS: System parameter C
      14362 = 1 (Name=DYNSYS_PAR_C+2)  // FB2 FB DYNSYS: System parameter C
      14362 = 0 (Name=DYNSYS_PAR_C+2)  // FB2 FB DYNSYS: System parameter C
      14362 = 0 (Name=DYNSYS_PAR_C+2)  // FB2 FB DYNSYS: System parameter C
      14362 = 0 (Name=DYNSYS_PAR_C+2)  // FB2 FB DYNSYS: System parameter C
      14362 = 0 (Name=DYNSYS_PAR_C+2)  // FB2 FB DYNSYS: System parameter C
      14362 = 1 (Name=DYNSYS_PAR_C+2)  // FB2 FB DYNSYS: System parameter C
      14410 = 216 (Name=DYNSYS_IN1_PARID+2)  // FB0 FB DYNSYS: Parameter ID for input 1
      14338 = 1 (Name=DYNSYS_MODE+2)  // FB0 FB DYNSYS: Mode (note: set SCTRL_ADD_SET_PARID = DYNSYS_OUT1_VALUE+X for activation)
    DYNSYS+3:
      14339 = 0 (Name=DYNSYS_MODE+3)  // FB3 FB DYNSYS: Mode
      14347 = 0 (Name=DYNSYS_PAR_A+3)  // FB3 FB DYNSYS: System parameter A
      14347 = 0 (Name=DYNSYS_PAR_A+3)  // FB3 FB DYNSYS: System parameter A
      14347 = 0 (Name=DYNSYS_PAR_A+3)  // FB3 FB DYNSYS: System parameter A
      14347 = 0 (Name=DYNSYS_PAR_A+3)  // FB3 FB DYNSYS: System parameter A
      14347 = 1 (Name=DYNSYS_PAR_A+3)  // FB3 FB DYNSYS: System parameter A
      14347 = 0 (Name=DYNSYS_PAR_A+3)  // FB3 FB DYNSYS: System parameter A
      14347 = 0 (Name=DYNSYS_PAR_A+3)  // FB3 FB DYNSYS: System parameter A
      14347 = 0 (Name=DYNSYS_PAR_A+3)  // FB3 FB DYNSYS: System parameter A
      14347 = 0 (Name=DYNSYS_PAR_A+3)  // FB3 FB DYNSYS: System parameter A
      14347 = 1 (Name=DYNSYS_PAR_A+3)  // FB3 FB DYNSYS: System parameter A
      14347 = 0 (Name=DYNSYS_PAR_A+3)  // FB3 FB DYNSYS: System parameter A
      14347 = 0 (Name=DYNSYS_PAR_A+3)  // FB3 FB DYNSYS: System parameter A
      14347 = 0 (Name=DYNSYS_PAR_A+3)  // FB3 FB DYNSYS: System parameter A
      14347 = 0 (Name=DYNSYS_PAR_A+3)  // FB3 FB DYNSYS: System parameter A
      14347 = 1 (Name=DYNSYS_PAR_A+3)  // FB3 FB DYNSYS: System parameter A
      14347 = 0 (Name=DYNSYS_PAR_A+3)  // FB3 FB DYNSYS: System parameter A
      14355 = 1 (Name=DYNSYS_PAR_B+3)  // FB3 FB DYNSYS: System parameter B
      14355 = 0 (Name=DYNSYS_PAR_B+3)  // FB3 FB DYNSYS: System parameter B
      14355 = 0 (Name=DYNSYS_PAR_B+3)  // FB3 FB DYNSYS: System parameter B
      14355 = 0 (Name=DYNSYS_PAR_B+3)  // FB3 FB DYNSYS: System parameter B
      14363 = 1 (Name=DYNSYS_PAR_C+3)  // FB3 FB DYNSYS: System parameter C
      14363 = 0 (Name=DYNSYS_PAR_C+3)  // FB3 FB DYNSYS: System parameter C
      14363 = 0 (Name=DYNSYS_PAR_C+3)  // FB3 FB DYNSYS: System parameter C
      14363 = 0 (Name=DYNSYS_PAR_C+3)  // FB3 FB DYNSYS: System parameter C
      14363 = 0 (Name=DYNSYS_PAR_C+3)  // FB3 FB DYNSYS: System parameter C
      14363 = 1 (Name=DYNSYS_PAR_C+3)  // FB3 FB DYNSYS: System parameter C
      14363 = 0 (Name=DYNSYS_PAR_C+3)  // FB3 FB DYNSYS: System parameter C
      14363 = 0 (Name=DYNSYS_PAR_C+3)  // FB3 FB DYNSYS: System parameter C
      14411 = 214 (Name=DYNSYS_IN1_PARID+3)  // FB3 FB DYNSYS: Parameter ID for input 1
      14339 = 1 (Name=DYNSYS_MODE+3)  // FB3 FB DYNSYS: Mode
    DYNSYS+4:
      14340 = 0 (Name=DYNSYS_MODE+4)  // FB4 FB DYNSYS: Mode
      14348 = 0 (Name=DYNSYS_PAR_A+4)  // FB4 FB DYNSYS: System parameter A
      14348 = 0 (Name=DYNSYS_PAR_A+4)  // FB4 FB DYNSYS: System parameter A
      14348 = 0 (Name=DYNSYS_PAR_A+4)  // FB4 FB DYNSYS: System parameter A
      14348 = 0 (Name=DYNSYS_PAR_A+4)  // FB4 FB DYNSYS: System parameter A
      14348 = 1 (Name=DYNSYS_PAR_A+4)  // FB4 FB DYNSYS: System parameter A
      14348 = 0 (Name=DYNSYS_PAR_A+4)  // FB4 FB DYNSYS: System parameter A
      14348 = 0 (Name=DYNSYS_PAR_A+4)  // FB4 FB DYNSYS: System parameter A
      14348 = 0 (Name=DYNSYS_PAR_A+4)  // FB4 FB DYNSYS: System parameter A
      14348 = 0 (Name=DYNSYS_PAR_A+4)  // FB4 FB DYNSYS: System parameter A
      14348 = 1 (Name=DYNSYS_PAR_A+4)  // FB4 FB DYNSYS: System parameter A
      14348 = 0 (Name=DYNSYS_PAR_A+4)  // FB4 FB DYNSYS: System parameter A
      14348 = 0 (Name=DYNSYS_PAR_A+4)  // FB4 FB DYNSYS: System parameter A
      14348 = 0 (Name=DYNSYS_PAR_A+4)  // FB4 FB DYNSYS: System parameter A
      14348 = 0 (Name=DYNSYS_PAR_A+4)  // FB4 FB DYNSYS: System parameter A
      14348 = 1 (Name=DYNSYS_PAR_A+4)  // FB4 FB DYNSYS: System parameter A
      14348 = 0 (Name=DYNSYS_PAR_A+4)  // FB4 FB DYNSYS: System parameter A
      14356 = 1 (Name=DYNSYS_PAR_B+4)  // FB4 FB DYNSYS: System parameter B
      14356 = 0 (Name=DYNSYS_PAR_B+4)  // FB4 FB DYNSYS: System parameter B
      14356 = 0 (Name=DYNSYS_PAR_B+4)  // FB4 FB DYNSYS: System parameter B
      14356 = 0 (Name=DYNSYS_PAR_B+4)  // FB4 FB DYNSYS: System parameter B
      14364 = 0 (Name=DYNSYS_PAR_C+4)  // FB4 FB DYNSYS: System parameter C
      14364 = 0 (Name=DYNSYS_PAR_C+4)  // FB4 FB DYNSYS: System parameter C
      14364 = 1 (Name=DYNSYS_PAR_C+4)  // FB4 FB DYNSYS: System parameter C
      14364 = 0 (Name=DYNSYS_PAR_C+4)  // FB4 FB DYNSYS: System parameter C
      14364 = 0 (Name=DYNSYS_PAR_C+4)  // FB4 FB DYNSYS: System parameter C
      14364 = 0 (Name=DYNSYS_PAR_C+4)  // FB4 FB DYNSYS: System parameter C
      14364 = 0 (Name=DYNSYS_PAR_C+4)  // FB4 FB DYNSYS: System parameter C
      14364 = 1 (Name=DYNSYS_PAR_C+4)  // FB4 FB DYNSYS: System parameter C
      14412 = 214 (Name=DYNSYS_IN1_PARID+4)  // FB4 FB DYNSYS: Parameter ID for input 1
      14340 = 1 (Name=DYNSYS_MODE+4)  // FB4 FB DYNSYS: Mode
    COUNT:
      13856 = 0 (Name=COUNT_SET_VALUE+0)  // FB0 COUNT: Value to set counter
      13864 = 3 (Name=COUNT_MAX_VALUE+0)  // FB0 COUNT: Maximum counter value
      13872 = 3 (Name=COUNT_CMP_VALUE+0)  // FB0 COUNT: Comparator compare value
      13824 = 2 (Name=COUNT_MODE+0)  // FB0 COUNT: Mode
```

### Data object Logical/gAxisVibLobj/gAxisVibLi (Ax)

#### gAxisVibLi.ax
```
InitParameter (Version=5.12.2, NcSwId=Acp10)
  ACP10AXIS_typ:
    dig_in:
      level:
        reference = ncACTIV_HI
        pos_hw_end = ncACTIV_HI
        neg_hw_end = ncACTIV_HI
        trigger1 = ncACTIV_HI
        trigger2 = ncACTIV_HI
    encoder_if:
      parameter:
        count_dir = ncSTANDARD
        scaling:
          load:
            units = 1000
            rev_motor = 1
    limit:
      parameter:
        v_pos = 54000.0
        v_neg = 54000.0
        a1_pos = 5000000.0
        a2_pos = 5000000.0
        a1_neg = 5000000.0
        a2_neg = 5000000.0
        t_jolt = 0
        t_in_pos = 0
        pos_sw_end = 2000000000
        neg_sw_end = -2000000000
        ds_warning = 500
        ds_stop = 1000
        a_stop = 1.0e30
        dv_stop = 0
        dv_stop_mode = ncOFF
    controller:
      mode = ncUF
      position:
        kv = 50
        tn = 0
        t_predict = 0.0004
        t_total = 0.0004
        p_max = 1.0e30
        i_max = 0
      speed:
        kv = 2.0
        tn = 0
        t_filter = 0.0
        isq_filter1:
          type = ncOFF
          a0 = 0.0
          a1 = 0.0
          b0 = 0.0
          b1 = 0.0
          b2 = 0.0
          c0_par_id = 0
          c1_par_id = 0
        isq_filter2:
          type = ncOFF
          a0 = 0.0
          a1 = 0.0
          b0 = 0.0
          b1 = 0.0
          b2 = 0.0
          c0_par_id = 0
          c1_par_id = 0
        isq_filter3:
          type = ncOFF
          a0 = 0.0
          a1 = 0.0
          b0 = 0.0
          b1 = 0.0
          b2 = 0.0
          c0_par_id = 0
          c1_par_id = 0
      uf:
        type = ncLINEAR
        auto_config = ncOFF
        u0 = 0
        un = 0
        fn = 50.0
        k_f_slip = 0
      ff:
        mode = ncSTANDARD
        torque_load = 0.0
        torque_pos = 0.0
        torque_neg = 0.0
        kv_torque = 0.0
        inertia = 0.0
        t_filter_a = 0.0
      fb:
        mode = ncSTANDARD
        speed_mix_ratio = 0.0
        speed_kv = 2.0
      model:
        mass1:
          inertia = 0
          viscous_friction = 0
        mass2:
          inertia = 0
          viscous_friction = 0
          stiffness = 0
          damping = 0
    move:
      stop:
        parameter[0]:
          decel_ramp = ncA_LIMIT
          controller = ncON
        parameter[1]:
          decel_ramp = ncA_LIMIT
          controller = ncON
        parameter[2]:
          decel_ramp = ncA_LIMIT
          controller = ncON
        parameter[3]:
          decel_ramp = ncA_LIMIT
          controller = ncON
        quickstop:
          decel_ramp = ncA_LIMIT
          t_jolt = 0
        drive_error:
          decel_ramp = ncA_LIMIT
      homing:
        parameter:
          s = 0
          v_switch = 5000
          v_trigger = 500
          a = 50000
          mode = ncDIRECT
          edge_sw = ncPOSITIVE
          start_dir = ncPOSITIVE
          trigg_dir = ncPOSITIVE
          ref_pulse = ncOFF
          fix_dir = ncOFF
          tr_s_block = 0
          torque_lim = 0
          ds_block = 0
          ds_stop = 0
      basis:
        parameter:
          v_pos = 50000.0
          v_neg = 50000.0
          a1_pos = 500000.0
          a2_pos = 500000.0
          a1_neg = 500000.0
          a2_neg = 500000.0
    message:
      text:
        parameter:
          format = ncBREAK + ncZERO
          columns = 80
          data_modul = acp10etxen
```

### Data object Logical/gAxisVibLobj/lfCurCtr (Apt)

#### lfCurCtr.apt
```
AcoposParameterTable:
  Root Parameters:
    128 = 1 (Name=SGEN_SW_END_IGNORE)  // Limit values: Ignore SW end positions
    652 = 0 (Name=MOTOR_ENCOD_ATTR)  // Motor: Encoder: Attribute
    1215 = 0 (Name=MOTOR_TEMPSENS_TYPE)  // Temperature sensor: Type
    90 = 76 (Name=BRAKE_MODE)  // Motor holding brake: Mode
    1208 = 1 (Name=MOTOR_NUM_PHASES)  // Motor: Number of motor phases
    Axis Parameter Identification, Synchronous Motor:
      Group  // General Parameters
        30 = 2 (Name=MOTOR_TYPE)  // Motor: Type
        31 = 0x0203 (Name=MOTOR_COMPATIBILITY)  // Motor: Software compatibility
        46 = 1 (Name=MOTOR_WIND_CONNECT)  // Motor: Winding connection
        62 = 0 (Name=MOTOR_INERTIA, Unit=kgm²)  // Motor: Moment of inertia
        849 = 0 (Name=MOTOR_TAU_THERM, Unit=s)  // Motor: Thermal time constant
      Group  // Brake Parameters
        42 = 0 (Name=MOTOR_BRAKE_CURR_RATED, Unit=A)  // Motor holding brake: Rated current
        43 = 0 (Name=MOTOR_BRAKE_TORQ_RATED, Unit=Nm)  // Motor holding brake: Rated torque
        44 = 0 (Name=MOTOR_BRAKE_ON_TIME, Unit=s)  // Motor holding brake: Engaging delay
        45 = 0 (Name=MOTOR_BRAKE_OFF_TIME, Unit=s)  // Motor holding brake: Release delay
      Group  // Thermo Sensor Parameters
        64 = 0 (Name=MOTOR_TEMPSENS_PAR1)  // Temperature sensor: Parameter 1
        65 = 0 (Name=MOTOR_TEMPSENS_PAR2)  // Temperature sensor: Parameter 2
        66 = 0 (Name=MOTOR_TEMPSENS_PAR3)  // Temperature sensor: Parameter 3
        67 = 0 (Name=MOTOR_TEMPSENS_PAR4)  // Temperature sensor: Parameter 4
        68 = 0 (Name=MOTOR_TEMPSENS_PAR5)  // Temperature sensor: Parameter 5
        69 = 0 (Name=MOTOR_TEMPSENS_PAR6)  // Temperature sensor: Parameter 6
        70 = 0 (Name=MOTOR_TEMPSENS_PAR7)  // Temperature sensor: Parameter 7
        71 = 0 (Name=MOTOR_TEMPSENS_PAR8)  // Temperature sensor: Parameter 8
        72 = 0 (Name=MOTOR_TEMPSENS_PAR9)  // Temperature sensor: Parameter 9
        73 = 0 (Name=MOTOR_TEMPSENS_PAR10)  // Temperature sensor: Parameter 10
        74 = 50 (Name=MOTOR_WIND_TEMP_MAX, Unit=°C)  // Temperature sensor: Limit temperature
      Group  // Result Parameters of Parameter Identification
        47 = 1 (Name=MOTOR_POLEPAIRS)  // Motor: Number of pole-pairs
        48 = 200 (Name=MOTOR_VOLTAGE_RATED, Unit=V)  // Motor: Rated voltage
        50 = 6000 (Name=MOTOR_SPEED_RATED, Unit=1/min)  // Motor: Rated speed
        51 = 6600 (Name=MOTOR_SPEED_MAX, Unit=1/min)  // Motor: Maximum speed
        52 = 1 (Name=MOTOR_TORQ_STALL, Unit=Nm)  // Motor: Stall torque
        53 = 1 (Name=MOTOR_TORQ_RATED, Unit=Nm)  // Motor: Rated torque
        54 = 1 (Name=MOTOR_TORQ_MAX, Unit=Nm)  // Motor: Peak torque
        56 = 1 (Name=MOTOR_CURR_STALL, Unit=A)  // Motor: Stall current
        57 = 2.6 (Name=MOTOR_CURR_RATED, Unit=A)  // Motor: Rated current
        58 = 3 (Name=MOTOR_CURR_MAX, Unit=A)  // Motor: Peak current
        59 = 1 (Name=MOTOR_WIND_CROSS_SECT, Unit=mm²)  // Motor: Line cross section
        60 = 92.617 (Name=MOTOR_STATOR_RESISTANCE, Unit=Ohm)  // Motor: Stator resistance
        61 = 5.803 (Name=MOTOR_STATOR_INDUCTANCE, Unit=Henry)  // Motor: Stator inductance
        1208 = 1 (Name=MOTOR_NUM_PHASES)  // Motor: Number of motor phases
      DELAY:
        777 = DELAY_TIME+0 (Name=FUNCTION_BLOCK_CREATE)  // Function block: Create a FB instance
        7168 = CYCLIC_TODRV_COUNT (Name=DELAY_IN_PARID+0)  // FB0 DELAY parameter ID of input
        7176 = 0.0004 (Name=DELAY_TIME+0, Unit=s)  // FB0 DELAY time
      COUNT:
        777 = COUNT_MODE+0 (Name=FUNCTION_BLOCK_CREATE)  // Function block: Create a FB instance
        585 = 300 (Name=USER_I4_VAR2)  // Function block: User I4 variable2
        13824 = 0 (Name=COUNT_MODE+0)  // FB0 COUNT: Mode
        13904 = CONST_I4_ONE (Name=COUNT_ENABLE_PARID+0)  // FB0 COUNT: Parameter ID of enable input
        13832 = CYCLIC_TODRV_COUNT (Name=COUNT_EV1_PARID+0)  // FB0 COUNT: Parameter ID of event input1
        13840 = DELAY_VALUE_I4+0 (Name=COUNT_EV2_PARID+0)  // FB0 COUNT: Parameter ID of event input2
        13872 = 2 (Name=COUNT_CMP_VALUE+0)  // FB0 FB COUNT: Comparator compare value
        13864 = 3 (Name=COUNT_MAX_VALUE+0)  // FB0 COUNT: Maximum counter value
        13824 = 5 (Name=COUNT_MODE+0)  // FB0 COUNT: Mode
      CMP:
        777 = CMP_MODE+0 (Name=FUNCTION_BLOCK_CREATE)  // Function block: Create a FB instance
        6656 = COUNT_VALUE+0 (Name=CMP_IN_PARID+0)  // FB0 CMP parameter ID of input
        6664 = 2 (Name=CMP_THRESHOLD+0)  // FB0 CMP threshold
        6688 = 6 (Name=CMP_MODE+0)  // FB0 CMP mode
      Group:
        232 = 0 (Name=CYCLIC_TODRV_PAR_INDEX)  // Cyclic communication: Parameter index of data to drive
        207 = CYCLIC_FRDRV_REC_INDEX (Name=CYCLIC_TODRV_PARID)  // Cyclic communication: Parameter ID of data to drive
        777 = IPL_MODE+0 (Name=FUNCTION_BLOCK_CREATE, Disabled=FALSE)  // Function block: Create a FB instance
        8712 = USER_R4_VAR1 (Name=IPL_IN_PARID+0, Disabled=FALSE)  // FB0 FB IPL: Parameter ID of input
        8760 = CMP_VALUE+0 (Name=IPL_EV_PARID+0)  // FB0 FB IPL: Parameter ID of event input
        8720 = 1600 (Name=IPL_CYCLE_TIME+0, Unit=us)  // FB0 FB IPL: Cycle time
        8704 = 2 (Name=IPL_MODE+0, Disabled=FALSE)  // FB0 FB IPL: Mode - (4) quadric no overshoot
      Group:
        347 = 10000 (Name=F_SWITCH, Unit=cps)  // Inverter: Switch frequency
        49 = 100 (Name=MOTOR_VOLTAGE_CONST, Unit=mV*min)  // Motor: Voltage constant
        813 = 0  // PARID_SIGEN_OFFS
        55 = 3 (Name=MOTOR_TORQ_CONST, Unit=Nm/A)  // Motor: Torque constant
        63 = 0 (Name=MOTOR_COMMUT_OFFSET, Unit=rad)  // Motor: Commutation offset
        328 = 5 (Name=CONTROLLER_MODE)  // CTRL Controller: Mode
        713 = 8752 (Name=ICTRL_SET_PARID)  // CTRL Current controller: Set value parameter ID of stator current quadrature component
        1480 = 0 (Name=TLIM_MODE)  // CTRL Torque limiter: Mode
        1569 = 2451 (Name=ICTRL_US_FILTER1_A0)  // CTRL Current: Set voltage filter coefficient A0
        1570 = 2200 (Name=ICTRL_US_FILTER1_A1)  // CTRL Current: Set voltage filter coefficient A1
        1568 = 1 (Name=ICTRL_US_FILTER_TYPE)  // CTRL Current: Set voltage filter type
        1166 = 0 (Name=ICTRL_AUTO_CONFIG)  // CTRL Current: Automatic configuration
        223 = 2000 (Name=ICTRL_KV, Unit=V/A)  // CTRL Current controller: Proportional amplification factor
        225 = 0.0033906708 (Name=ICTRL_TI, Unit=s)  // CTRL Current controller: Integral action time
```

### Data object Logical/gAxisVibLobj/lfNew (Apt)

#### lfNew.apt
```
AcoposParameterTable:
  Root Parameters:
    128 = 1 (Name=SGEN_SW_END_IGNORE)  // Limit values: Ignore SW end positions
    652 = 0 (Name=MOTOR_ENCOD_ATTR)  // Motor: Encoder: Attribute
    1215 = 0 (Name=MOTOR_TEMPSENS_TYPE)  // Temperature sensor: Type
    90 = 76 (Name=BRAKE_MODE)  // Motor holding brake: Mode
    1208 = 1 (Name=MOTOR_NUM_PHASES)  // Motor: Number of motor phases
    Axis Parameter Identification, Synchronous Motor:
      Group  // General Parameters
        30 = 2 (Name=MOTOR_TYPE)  // Motor: Type
        31 = 0x0203 (Name=MOTOR_COMPATIBILITY)  // Motor: Software compatibility
        46 = 1 (Name=MOTOR_WIND_CONNECT)  // Motor: Winding connection
        62 = 0 (Name=MOTOR_INERTIA, Unit=kgm²)  // Motor: Moment of inertia
        849 = 0 (Name=MOTOR_TAU_THERM, Unit=s)  // Motor: Thermal time constant
      Group  // Brake Parameters
        42 = 0 (Name=MOTOR_BRAKE_CURR_RATED, Unit=A)  // Motor holding brake: Rated current
        43 = 0 (Name=MOTOR_BRAKE_TORQ_RATED, Unit=Nm)  // Motor holding brake: Rated torque
        44 = 0 (Name=MOTOR_BRAKE_ON_TIME, Unit=s)  // Motor holding brake: Engaging delay
        45 = 0 (Name=MOTOR_BRAKE_OFF_TIME, Unit=s)  // Motor holding brake: Release delay
      Group  // Thermo Sensor Parameters
        64 = 0 (Name=MOTOR_TEMPSENS_PAR1)  // Temperature sensor: Parameter 1
        65 = 0 (Name=MOTOR_TEMPSENS_PAR2)  // Temperature sensor: Parameter 2
        66 = 0 (Name=MOTOR_TEMPSENS_PAR3)  // Temperature sensor: Parameter 3
        67 = 0 (Name=MOTOR_TEMPSENS_PAR4)  // Temperature sensor: Parameter 4
        68 = 0 (Name=MOTOR_TEMPSENS_PAR5)  // Temperature sensor: Parameter 5
        69 = 0 (Name=MOTOR_TEMPSENS_PAR6)  // Temperature sensor: Parameter 6
        70 = 0 (Name=MOTOR_TEMPSENS_PAR7)  // Temperature sensor: Parameter 7
        71 = 0 (Name=MOTOR_TEMPSENS_PAR8)  // Temperature sensor: Parameter 8
        72 = 0 (Name=MOTOR_TEMPSENS_PAR9)  // Temperature sensor: Parameter 9
        73 = 0 (Name=MOTOR_TEMPSENS_PAR10)  // Temperature sensor: Parameter 10
        74 = 50 (Name=MOTOR_WIND_TEMP_MAX, Unit=°C)  // Temperature sensor: Limit temperature
      Group  // Result Parameters of Parameter Identification
        47 = 1 (Name=MOTOR_POLEPAIRS)  // Motor: Number of pole-pairs
        48 = 200 (Name=MOTOR_VOLTAGE_RATED, Unit=V)  // Motor: Rated voltage
        50 = 6000 (Name=MOTOR_SPEED_RATED, Unit=1/min)  // Motor: Rated speed
        51 = 6600 (Name=MOTOR_SPEED_MAX, Unit=1/min)  // Motor: Maximum speed
        52 = 1 (Name=MOTOR_TORQ_STALL, Unit=Nm)  // Motor: Stall torque
        53 = 1 (Name=MOTOR_TORQ_RATED, Unit=Nm)  // Motor: Rated torque
        54 = 1 (Name=MOTOR_TORQ_MAX, Unit=Nm)  // Motor: Peak torque
        56 = 1 (Name=MOTOR_CURR_STALL, Unit=A)  // Motor: Stall current
        58 = 0.2 (Name=MOTOR_CURR_MAX, Unit=A)  // Motor: Peak current
        57 = 0.15 (Name=MOTOR_CURR_RATED, Unit=A)  // Motor: Rated current
        59 = 1 (Name=MOTOR_WIND_CROSS_SECT, Unit=mm²)  // Motor: Line cross section
        60 = 92.617 (Name=MOTOR_STATOR_RESISTANCE, Unit=Ohm)  // Motor: Stator resistance
        61 = 5.803 (Name=MOTOR_STATOR_INDUCTANCE, Unit=Henry)  // Motor: Stator inductance
        1208 = 1 (Name=MOTOR_NUM_PHASES)  // Motor: Number of motor phases
      IPL:
        777 = IPL_MODE+0 (Name=FUNCTION_BLOCK_CREATE, Disabled=FALSE)  // Function block: Create a FB instance
        8712 = USER_R4_VAR1 (Name=IPL_IN_PARID+0, Disabled=FALSE)  // FB0 FB IPL: Parameter ID of input
        8760 = CYCLIC_TODRV_COUNT (Name=IPL_EV_PARID+0)  // FB0 FB IPL: Parameter ID of event input
        8720 = 800 (Name=IPL_CYCLE_TIME+0, Unit=us)  // FB0 FB IPL: Cycle time
        8704 = 2 (Name=IPL_MODE+0, Disabled=FALSE)  // FB0 FB IPL: Mode - (4) quadric no overshoot
      Group:
        347 = 10000 (Name=F_SWITCH, Unit=cps)  // Inverter: Switch frequency
        49 = 100 (Name=MOTOR_VOLTAGE_CONST, Unit=mV*min)  // Motor: Voltage constant
        813 = 0  // PARID_SIGEN_OFFS
        55 = 3 (Name=MOTOR_TORQ_CONST, Unit=Nm/A)  // Motor: Torque constant
        63 = 0 (Name=MOTOR_COMMUT_OFFSET, Unit=rad)  // Motor: Commutation offset
        713 = 8752 (Name=ICTRL_SET_PARID)  // CTRL Current controller: Set value parameter ID of stator current quadrature component
        1480 = 0 (Name=TLIM_MODE)  // CTRL Torque limiter: Mode
        1569 = 2451 (Name=ICTRL_US_FILTER1_A0)  // CTRL Current: Set voltage filter coefficient A0
        1570 = 2200 (Name=ICTRL_US_FILTER1_A1)  // CTRL Current: Set voltage filter coefficient A1
        1568 = 1 (Name=ICTRL_US_FILTER_TYPE)  // CTRL Current: Set voltage filter type
        1166 = 0 (Name=ICTRL_AUTO_CONFIG)  // CTRL Current: Automatic configuration
        223 = 2000 (Name=ICTRL_KV, Unit=V/A)  // CTRL Current controller: Proportional amplification factor
        225 = 0.0033906708 (Name=ICTRL_TI, Unit=s)  // CTRL Current controller: Integral action time
        328 = 5 (Name=CONTROLLER_MODE)  // CTRL Controller: Mode
      Voltage observer:
        1354 = 1 (Name=OBS_MODE_BITS)  // Observer: Mode bits
        1298 = 25.4481 (Name=OBS_VOLT_INVCL_A1)  // Voltage observer: Inverter adjustment amplification factor
        1299 = 2.2113 (Name=OBS_VOLT_INVCL_A2, Unit=1/A)  // Voltage observer: Inverter adjustment exponent
        232 = 0 (Name=CYCLIC_TODRV_PAR_INDEX)  // Cyclic communication: Parameter index of data to drive
    207 = CYCLIC_FRDRV_REC_INDEX (Name=CYCLIC_TODRV_PARID)  // Cyclic communication: Parameter ID of data to drive
    777 = ARITH_MODE+0 (Name=FUNCTION_BLOCK_CREATE)  // Function block: Create a FB instance
    777 = DYNSYS_MODE+0 (Name=FUNCTION_BLOCK_CREATE)  // Function block: Create a FB instance
    777 = ARITH_MODE+1 (Name=FUNCTION_BLOCK_CREATE)  // Function block: Create a FB instance
    777 = ARITH_MODE+2 (Name=FUNCTION_BLOCK_CREATE)  // Function block: Create a FB instance
    777 = DYNSYS_MODE+1 (Name=FUNCTION_BLOCK_CREATE)  // Function block: Create a FB instance
    777 = DYNSYS_MODE+2 (Name=FUNCTION_BLOCK_CREATE)  // Function block: Create a FB instance
    777 = DYNSYS_MODE+3 (Name=FUNCTION_BLOCK_CREATE)  // Function block: Create a FB instance
    777 = DYNSYS_MODE+4 (Name=FUNCTION_BLOCK_CREATE)  // Function block: Create a FB instance
    777 = VAR_I4_0+0 (Name=FUNCTION_BLOCK_CREATE)  // Function block: Create a FB instance
    777 = VAR_R4_0+0 (Name=FUNCTION_BLOCK_CREATE)  // Function block: Create a FB instance
    777 = MINMAX_MODE+0 (Name=FUNCTION_BLOCK_CREATE)  // Function block: Create a FB instance
    777 = MINMAX_MODE+1 (Name=FUNCTION_BLOCK_CREATE)  // Function block: Create a FB instance
    777 = COUNT_MODE+0 (Name=FUNCTION_BLOCK_CREATE)  // Function block: Create a FB instance
    777 = FILTER_MODE+0 (Name=FUNCTION_BLOCK_CREATE)  // Function block: Create a FB instance
    ARITH EMF:
      3584 = 0 (Name=ARITH_MODE+0)  // FB0 ARITH Mode
      3592 = 216 (Name=ARITH_IN1_PARID+0)  // FB0 ARITH Parameter ID of input1
      3600 = 214 (Name=ARITH_IN2_PARID+0)  // FB0 ARITH Parameter ID of input2
      3632 = 1 (Name=ARITH_K1+0)  // FB0 ARITH Multiplication factor1
      3640 = -4.2 (Name=ARITH_K2+0)  // FB0 ARITH Multiplication factor2
      3584 = 4 (Name=ARITH_MODE+0)  // FB0 ARITH Mode
    DYNSYS Integrate EMF:
      14336 = 0 (Name=DYNSYS_MODE+0)  // FB0 FB DYNSYS: Mode
      14344 = 0.99 (Name=DYNSYS_PAR_A+0)  // FB0 FB DYNSYS: System parameter A
      14344 = 0.0002 (Name=DYNSYS_PAR_A+0)  // FB0 FB DYNSYS: System parameter A
      14344 = 0 (Name=DYNSYS_PAR_A+0)  // FB0 FB DYNSYS: System parameter A
      14344 = 0 (Name=DYNSYS_PAR_A+0)  // FB0 FB DYNSYS: System parameter A
      14344 = 0 (Name=DYNSYS_PAR_A+0)  // FB0 FB DYNSYS: System parameter A
      14344 = 0 (Name=DYNSYS_PAR_A+0)  // FB0 FB DYNSYS: System parameter A
      14344 = 0 (Name=DYNSYS_PAR_A+0)  // FB0 FB DYNSYS: System parameter A
      14344 = 0 (Name=DYNSYS_PAR_A+0)  // FB0 FB DYNSYS: System parameter A
      14344 = 0 (Name=DYNSYS_PAR_A+0)  // FB0 FB DYNSYS: System parameter A
      14352 = 0.0002 (Name=DYNSYS_PAR_B+0)  // FB0 FB DYNSYS: System parameter B
      14352 = 0 (Name=DYNSYS_PAR_B+0)  // FB0 FB DYNSYS: System parameter B
      14352 = 1 (Name=DYNSYS_PAR_B+0)  // FB0 FB DYNSYS: System parameter B
      14352 = 0 (Name=DYNSYS_PAR_B+0)  // FB0 FB DYNSYS: System parameter B
      14352 = 0 (Name=DYNSYS_PAR_B+0)  // FB0 FB DYNSYS: System parameter B
      14352 = 1 (Name=DYNSYS_PAR_B+0)  // FB0 FB DYNSYS: System parameter B
      14360 = 1 (Name=DYNSYS_PAR_C+0)  // FB0 FB DYNSYS: System parameter C
      14360 = 0 (Name=DYNSYS_PAR_C+0)  // FB0 FB DYNSYS: System parameter C
      14360 = 0 (Name=DYNSYS_PAR_C+0)  // FB0 FB DYNSYS: System parameter C
      14360 = 0 (Name=DYNSYS_PAR_C+0)  // FB0 FB DYNSYS: System parameter C
      14360 = 0 (Name=DYNSYS_PAR_C+0)  // FB0 FB DYNSYS: System parameter C
      14360 = 1 (Name=DYNSYS_PAR_C+0)  // FB0 FB DYNSYS: System parameter C
      14408 = ARITH_VALUE_R4+0 (Name=DYNSYS_IN1_PARID+0)  // FB0 FB DYNSYS: Parameter ID for input 1
      14416 = 214 (Name=DYNSYS_IN2_PARID+0)  // FB0 FB DYNSYS: Parameter ID for input 2
      14336 = 1 (Name=DYNSYS_MODE+0)  // FB0 FB DYNSYS: Mode (note: set SCTRL_ADD_SET_PARID = DYNSYS_OUT1_VALUE+X for activation)
    ARITH Airgap:
      3585 = 0 (Name=ARITH_MODE+1)  // FB0 ARITH Mode
      3593 = DYNSYS_OUT2_VALUE+0 (Name=ARITH_IN1_PARID+1)  // FB0 ARITH Parameter ID of input1
      3601 = DYNSYS_OUT1_VALUE+0 (Name=ARITH_IN2_PARID+1)  // FB0 ARITH Parameter ID of input2
      3585 = 5 (Name=ARITH_MODE+1)  // FB0 ARITH Mode
    ARITH Observer:
      3586 = 0 (Name=ARITH_MODE+2)  // FB2 FB ARITH: Mode
      3594 = 1296 (Name=ARITH_IN1_PARID+2)  // FB2 FB ARITH: Parameter ID of input1
      3602 = 1297 (Name=ARITH_IN2_PARID+2)  // FB2 FB ARITH: Parameter ID of input2
      3586 = 2 (Name=ARITH_MODE+2)  // FB2 FB ARITH: Mode
    DYNSYS+1:
      14337 = 0 (Name=DYNSYS_MODE+1)  // FB0 FB DYNSYS: Mode
      14345 = 0 (Name=DYNSYS_PAR_A+1)  // FB0 FB DYNSYS: System parameter A
      14345 = 0 (Name=DYNSYS_PAR_A+1)  // FB0 FB DYNSYS: System parameter A
      14345 = 0 (Name=DYNSYS_PAR_A+1)  // FB0 FB DYNSYS: System parameter A
      14345 = 0 (Name=DYNSYS_PAR_A+1)  // FB0 FB DYNSYS: System parameter A
      14345 = 1 (Name=DYNSYS_PAR_A+1)  // FB0 FB DYNSYS: System parameter A
      14345 = 0 (Name=DYNSYS_PAR_A+1)  // FB0 FB DYNSYS: System parameter A
      14345 = 0 (Name=DYNSYS_PAR_A+1)  // FB0 FB DYNSYS: System parameter A
      14345 = 0 (Name=DYNSYS_PAR_A+1)  // FB0 FB DYNSYS: System parameter A
      14345 = 0 (Name=DYNSYS_PAR_A+1)  // FB0 FB DYNSYS: System parameter A
      14345 = 1 (Name=DYNSYS_PAR_A+1)  // FB0 FB DYNSYS: System parameter A
      14345 = 0 (Name=DYNSYS_PAR_A+1)  // FB0 FB DYNSYS: System parameter A
      14345 = 0 (Name=DYNSYS_PAR_A+1)  // FB0 FB DYNSYS: System parameter A
      14345 = 0 (Name=DYNSYS_PAR_A+1)  // FB0 FB DYNSYS: System parameter A
      14345 = 0 (Name=DYNSYS_PAR_A+1)  // FB0 FB DYNSYS: System parameter A
      14345 = 1 (Name=DYNSYS_PAR_A+1)  // FB0 FB DYNSYS: System parameter A
      14345 = 0 (Name=DYNSYS_PAR_A+1)  // FB0 FB DYNSYS: System parameter A
      14353 = 1 (Name=DYNSYS_PAR_B+1)  // FB1 FB DYNSYS: System parameter B
      14353 = 0 (Name=DYNSYS_PAR_B+1)  // FB1 FB DYNSYS: System parameter B
      14353 = 0 (Name=DYNSYS_PAR_B+1)  // FB1 FB DYNSYS: System parameter B
      14353 = 0 (Name=DYNSYS_PAR_B+1)  // FB1 FB DYNSYS: System parameter B
      14361 = 1 (Name=DYNSYS_PAR_C+1)  // FB1 FB DYNSYS: System parameter C
      14361 = 0 (Name=DYNSYS_PAR_C+1)  // FB1 FB DYNSYS: System parameter C
      14361 = 0 (Name=DYNSYS_PAR_C+1)  // FB1 FB DYNSYS: System parameter C
      14361 = 0 (Name=DYNSYS_PAR_C+1)  // FB1 FB DYNSYS: System parameter C
      14361 = 0 (Name=DYNSYS_PAR_C+1)  // FB1 FB DYNSYS: System parameter C
      14361 = 1 (Name=DYNSYS_PAR_C+1)  // FB1 FB DYNSYS: System parameter C
      14361 = 0 (Name=DYNSYS_PAR_C+1)  // FB1 FB DYNSYS: System parameter C
      14361 = 0 (Name=DYNSYS_PAR_C+1)  // FB1 FB DYNSYS: System parameter C
      14409 = 216 (Name=DYNSYS_IN1_PARID+1)  // FB0 FB DYNSYS: Parameter ID for input 1
      14337 = 1 (Name=DYNSYS_MODE+1)  // FB0 FB DYNSYS: Mode (note: set SCTRL_ADD_SET_PARID = DYNSYS_OUT1_VALUE+X for activation)
    DYNSYS+2:
      14338 = 0 (Name=DYNSYS_MODE+2)  // FB0 FB DYNSYS: Mode
      14346 = 0 (Name=DYNSYS_PAR_A+2)  // FB0 FB DYNSYS: System parameter A
      14346 = 0 (Name=DYNSYS_PAR_A+2)  // FB0 FB DYNSYS: System parameter A
      14346 = 0 (Name=DYNSYS_PAR_A+2)  // FB0 FB DYNSYS: System parameter A
      14346 = 0 (Name=DYNSYS_PAR_A+2)  // FB0 FB DYNSYS: System parameter A
      14346 = 1 (Name=DYNSYS_PAR_A+2)  // FB0 FB DYNSYS: System parameter A
      14346 = 0 (Name=DYNSYS_PAR_A+2)  // FB0 FB DYNSYS: System parameter A
      14346 = 0 (Name=DYNSYS_PAR_A+2)  // FB0 FB DYNSYS: System parameter A
      14346 = 0 (Name=DYNSYS_PAR_A+2)  // FB0 FB DYNSYS: System parameter A
      14346 = 0 (Name=DYNSYS_PAR_A+2)  // FB0 FB DYNSYS: System parameter A
      14346 = 1 (Name=DYNSYS_PAR_A+2)  // FB0 FB DYNSYS: System parameter A
      14346 = 0 (Name=DYNSYS_PAR_A+2)  // FB0 FB DYNSYS: System parameter A
      14346 = 0 (Name=DYNSYS_PAR_A+2)  // FB0 FB DYNSYS: System parameter A
      14346 = 0 (Name=DYNSYS_PAR_A+2)  // FB0 FB DYNSYS: System parameter A
      14346 = 0 (Name=DYNSYS_PAR_A+2)  // FB0 FB DYNSYS: System parameter A
      14346 = 1 (Name=DYNSYS_PAR_A+2)  // FB0 FB DYNSYS: System parameter A
      14346 = 0 (Name=DYNSYS_PAR_A+2)  // FB0 FB DYNSYS: System parameter A
      14354 = 1 (Name=DYNSYS_PAR_B+2)  // FB2 FB DYNSYS: System parameter B
      14354 = 0 (Name=DYNSYS_PAR_B+2)  // FB2 FB DYNSYS: System parameter B
      14354 = 0 (Name=DYNSYS_PAR_B+2)  // FB2 FB DYNSYS: System parameter B
      14354 = 0 (Name=DYNSYS_PAR_B+2)  // FB2 FB DYNSYS: System parameter B
      14362 = 0 (Name=DYNSYS_PAR_C+2)  // FB2 FB DYNSYS: System parameter C
      14362 = 0 (Name=DYNSYS_PAR_C+2)  // FB2 FB DYNSYS: System parameter C
      14362 = 1 (Name=DYNSYS_PAR_C+2)  // FB2 FB DYNSYS: System parameter C
      14362 = 0 (Name=DYNSYS_PAR_C+2)  // FB2 FB DYNSYS: System parameter C
      14362 = 0 (Name=DYNSYS_PAR_C+2)  // FB2 FB DYNSYS: System parameter C
      14362 = 0 (Name=DYNSYS_PAR_C+2)  // FB2 FB DYNSYS: System parameter C
      14362 = 0 (Name=DYNSYS_PAR_C+2)  // FB2 FB DYNSYS: System parameter C
      14362 = 1 (Name=DYNSYS_PAR_C+2)  // FB2 FB DYNSYS: System parameter C
      14410 = 216 (Name=DYNSYS_IN1_PARID+2)  // FB0 FB DYNSYS: Parameter ID for input 1
      14338 = 1 (Name=DYNSYS_MODE+2)  // FB0 FB DYNSYS: Mode (note: set SCTRL_ADD_SET_PARID = DYNSYS_OUT1_VALUE+X for activation)
    DYNSYS+3:
      14339 = 0 (Name=DYNSYS_MODE+3)  // FB3 FB DYNSYS: Mode
      14347 = 0 (Name=DYNSYS_PAR_A+3)  // FB3 FB DYNSYS: System parameter A
      14347 = 0 (Name=DYNSYS_PAR_A+3)  // FB3 FB DYNSYS: System parameter A
      14347 = 0 (Name=DYNSYS_PAR_A+3)  // FB3 FB DYNSYS: System parameter A
      14347 = 0 (Name=DYNSYS_PAR_A+3)  // FB3 FB DYNSYS: System parameter A
      14347 = 1 (Name=DYNSYS_PAR_A+3)  // FB3 FB DYNSYS: System parameter A
      14347 = 0 (Name=DYNSYS_PAR_A+3)  // FB3 FB DYNSYS: System parameter A
      14347 = 0 (Name=DYNSYS_PAR_A+3)  // FB3 FB DYNSYS: System parameter A
      14347 = 0 (Name=DYNSYS_PAR_A+3)  // FB3 FB DYNSYS: System parameter A
      14347 = 0 (Name=DYNSYS_PAR_A+3)  // FB3 FB DYNSYS: System parameter A
      14347 = 1 (Name=DYNSYS_PAR_A+3)  // FB3 FB DYNSYS: System parameter A
      14347 = 0 (Name=DYNSYS_PAR_A+3)  // FB3 FB DYNSYS: System parameter A
      14347 = 0 (Name=DYNSYS_PAR_A+3)  // FB3 FB DYNSYS: System parameter A
      14347 = 0 (Name=DYNSYS_PAR_A+3)  // FB3 FB DYNSYS: System parameter A
      14347 = 0 (Name=DYNSYS_PAR_A+3)  // FB3 FB DYNSYS: System parameter A
      14347 = 1 (Name=DYNSYS_PAR_A+3)  // FB3 FB DYNSYS: System parameter A
      14347 = 0 (Name=DYNSYS_PAR_A+3)  // FB3 FB DYNSYS: System parameter A
      14355 = 1 (Name=DYNSYS_PAR_B+3)  // FB3 FB DYNSYS: System parameter B
      14355 = 0 (Name=DYNSYS_PAR_B+3)  // FB3 FB DYNSYS: System parameter B
      14355 = 0 (Name=DYNSYS_PAR_B+3)  // FB3 FB DYNSYS: System parameter B
      14355 = 0 (Name=DYNSYS_PAR_B+3)  // FB3 FB DYNSYS: System parameter B
      14363 = 1 (Name=DYNSYS_PAR_C+3)  // FB3 FB DYNSYS: System parameter C
      14363 = 0 (Name=DYNSYS_PAR_C+3)  // FB3 FB DYNSYS: System parameter C
      14363 = 0 (Name=DYNSYS_PAR_C+3)  // FB3 FB DYNSYS: System parameter C
      14363 = 0 (Name=DYNSYS_PAR_C+3)  // FB3 FB DYNSYS: System parameter C
      14363 = 0 (Name=DYNSYS_PAR_C+3)  // FB3 FB DYNSYS: System parameter C
      14363 = 1 (Name=DYNSYS_PAR_C+3)  // FB3 FB DYNSYS: System parameter C
      14363 = 0 (Name=DYNSYS_PAR_C+3)  // FB3 FB DYNSYS: System parameter C
      14363 = 0 (Name=DYNSYS_PAR_C+3)  // FB3 FB DYNSYS: System parameter C
      14411 = 8752 (Name=DYNSYS_IN1_PARID+3)  // FB3 FB DYNSYS: Parameter ID for input 1
      14339 = 1 (Name=DYNSYS_MODE+3)  // FB3 FB DYNSYS: Mode
    DYNSYS+4:
      14340 = 0 (Name=DYNSYS_MODE+4)  // FB4 FB DYNSYS: Mode
      14348 = 0 (Name=DYNSYS_PAR_A+4)  // FB4 FB DYNSYS: System parameter A
      14348 = 0 (Name=DYNSYS_PAR_A+4)  // FB4 FB DYNSYS: System parameter A
      14348 = 0 (Name=DYNSYS_PAR_A+4)  // FB4 FB DYNSYS: System parameter A
      14348 = 0 (Name=DYNSYS_PAR_A+4)  // FB4 FB DYNSYS: System parameter A
      14348 = 1 (Name=DYNSYS_PAR_A+4)  // FB4 FB DYNSYS: System parameter A
      14348 = 0 (Name=DYNSYS_PAR_A+4)  // FB4 FB DYNSYS: System parameter A
      14348 = 0 (Name=DYNSYS_PAR_A+4)  // FB4 FB DYNSYS: System parameter A
      14348 = 0 (Name=DYNSYS_PAR_A+4)  // FB4 FB DYNSYS: System parameter A
      14348 = 0 (Name=DYNSYS_PAR_A+4)  // FB4 FB DYNSYS: System parameter A
      14348 = 1 (Name=DYNSYS_PAR_A+4)  // FB4 FB DYNSYS: System parameter A
      14348 = 0 (Name=DYNSYS_PAR_A+4)  // FB4 FB DYNSYS: System parameter A
      14348 = 0 (Name=DYNSYS_PAR_A+4)  // FB4 FB DYNSYS: System parameter A
      14348 = 0 (Name=DYNSYS_PAR_A+4)  // FB4 FB DYNSYS: System parameter A
      14348 = 0 (Name=DYNSYS_PAR_A+4)  // FB4 FB DYNSYS: System parameter A
      14348 = 1 (Name=DYNSYS_PAR_A+4)  // FB4 FB DYNSYS: System parameter A
      14348 = 0 (Name=DYNSYS_PAR_A+4)  // FB4 FB DYNSYS: System parameter A
      14356 = 1 (Name=DYNSYS_PAR_B+4)  // FB4 FB DYNSYS: System parameter B
      14356 = 0 (Name=DYNSYS_PAR_B+4)  // FB4 FB DYNSYS: System parameter B
      14356 = 0 (Name=DYNSYS_PAR_B+4)  // FB4 FB DYNSYS: System parameter B
      14356 = 0 (Name=DYNSYS_PAR_B+4)  // FB4 FB DYNSYS: System parameter B
      14364 = 0 (Name=DYNSYS_PAR_C+4)  // FB4 FB DYNSYS: System parameter C
      14364 = 0 (Name=DYNSYS_PAR_C+4)  // FB4 FB DYNSYS: System parameter C
      14364 = 1 (Name=DYNSYS_PAR_C+4)  // FB4 FB DYNSYS: System parameter C
      14364 = 0 (Name=DYNSYS_PAR_C+4)  // FB4 FB DYNSYS: System parameter C
      14364 = 0 (Name=DYNSYS_PAR_C+4)  // FB4 FB DYNSYS: System parameter C
      14364 = 0 (Name=DYNSYS_PAR_C+4)  // FB4 FB DYNSYS: System parameter C
      14364 = 0 (Name=DYNSYS_PAR_C+4)  // FB4 FB DYNSYS: System parameter C
      14364 = 1 (Name=DYNSYS_PAR_C+4)  // FB4 FB DYNSYS: System parameter C
      14412 = 8752 (Name=DYNSYS_IN1_PARID+4)  // FB4 FB DYNSYS: Parameter ID for input 1
      14340 = 1 (Name=DYNSYS_MODE+4)  // FB4 FB DYNSYS: Mode
    COUNT:
      13856 = 0 (Name=COUNT_SET_VALUE+0)  // FB0 COUNT: Value to set counter
      13864 = 3 (Name=COUNT_MAX_VALUE+0)  // FB0 COUNT: Maximum counter value
      13872 = 3 (Name=COUNT_CMP_VALUE+0)  // FB0 COUNT: Comparator compare value
      13824 = 2 (Name=COUNT_MODE+0)  // FB0 COUNT: Mode
```

### Data object Logical/gAxisBeltobj/gAxisBelta (Apt)

#### gAxisBelta.apt
```
AcoposParameterTable:
  Root Parameters:
    128 = 1 (Name=SGEN_SW_END_IGNORE)  // Limit values: Ignore SW end positions
```

### Data object Logical/gAxisBeltobj/gAxisBelti (Ax)

#### gAxisBelti.ax
```
InitParameter (Version=5.23.1, NcSwId=ACP10)
  ACP10AXIS_typ:
    dig_in:
      level:
        reference = ncACTIV_HI
        pos_hw_end = ncACTIV_HI
        neg_hw_end = ncACTIV_HI
        trigger1 = ncACTIV_HI
        trigger2 = ncACTIV_HI
    encoder_if:
      parameter:
        count_dir = ncSTANDARD
        scaling:
          load:
            units = 107000
            rev_motor = 10
    limit:
      parameter:
        v_pos = 1000000.0
        v_neg = 1000000.0
        a1_pos = 1.0E+08
        a2_pos = 1.0E+08
        a1_neg = 1.0E+08
        a2_neg = 1.0E+08
        t_jolt = 0.08
        t_in_pos = 0.0
        pos_sw_end = 8388607
        neg_sw_end = -8388608
        ds_warning = 2000.0
        ds_stop = 2000.0
        a_stop = 1.0E+30
        dv_stop = 0.0
        dv_stop_mode = ncOFF
    controller:
      mode = ncPOSITION
      position:
        kv = 300.0
        tn = 0.0
        t_predict = 0.0004
        t_total = 0.0004
        p_max = 1.0E+30
        i_max = 2000.0
      speed:
        kv = 0.2
        tn = 0.0
        t_filter = 0.0
        isq_filter1:
          type = ncOFF
          a0 = 0.0
          a1 = 0.0
          b0 = 0.0
          b1 = 0.0
          b2 = 0.0
          c0_par_id = 0
          c1_par_id = 0
        isq_filter2:
          type = ncOFF
          a0 = 0.0
          a1 = 0.0
          b0 = 0.0
          b1 = 0.0
          b2 = 0.0
          c0_par_id = 0
          c1_par_id = 0
        isq_filter3:
          type = ncOFF
          a0 = 0.0
          a1 = 0.0
          b0 = 0.0
          b1 = 0.0
          b2 = 0.0
          c0_par_id = 0
          c1_par_id = 0
      uf:
        type = ncLINEAR + ncCORRECTION
        auto_config = ncMOTOR_PAR
        u0 = 0.0
        un = 0.0
        fn = 50.0
        k_f_slip = 0.0
      ff:
        mode = ncSTANDARD
        torque_load = 0.0
        torque_pos = 0.0
        torque_neg = 0.0
        kv_torque = 0.0
        inertia = 0.0
        t_filter_a = 0.0
      fb:
        mode = ncSTANDARD
        speed_mix_ratio = 0.0
        speed_kv = 0.0
      model:
        mass1:
          inertia = 0.0
          viscous_friction = 0.0
        mass2:
          inertia = 0.0
          viscous_friction = 0.0
          stiffness = 0.0
          damping = 0.0
    move:
      stop:
        parameter[0]:
          decel_ramp = ncA_LIMIT
          controller = ncON
        parameter[1]:
          decel_ramp = ncA_LIMIT
          controller = ncON
        parameter[2]:
          decel_ramp = ncA_LIMIT
          controller = ncON
        parameter[3]:
          decel_ramp = ncA_LIMIT
          controller = ncON
        quickstop:
          decel_ramp = ncA_LIMIT
          t_jolt = 0.0
        drive_error:
          decel_ramp = ncA_LIMIT
      homing:
        parameter:
          s = 0
          v_switch = 5000.0
          v_trigger = 500.0
          a = 50000.0
          mode = ncDIRECT
          edge_sw = ncPOSITIVE
          start_dir = ncPOSITIVE
          trigg_dir = ncPOSITIVE
          ref_pulse = ncOFF
          fix_dir = ncOFF
          tr_s_block = 0.0
          torque_lim = 0.0
          ds_block = 0.0
          ds_stop = 0.0
      basis:
        parameter:
          v_pos = 1000000.0
          v_neg = 1000000.0
          a1_pos = 1.0E+07
          a2_pos = 1.0E+07
          a1_neg = 1.0E+07
          a2_neg = 1.0E+07
    message:
      text:
        parameter:
          format = ncZERO
          columns = 81
          data_modul = acp10etxen
```

### Program Logical/vibratorCtrl

#### Variables.var
```iecst
VAR CONSTANT
	PI : REAL := 3.14159265359;
	CYCLE_TIME_s : REAL := 0.0008;
	PARID_IPL1_OUT : UINT := 8752;
	CONTROLLER_MODE_CURR_CTRL : UINT := 5;
END_VAR
VAR
	MC_Power_0 : MC_Power;
	Run : BOOL;
	amplitude_out : REAL;
	MaxCurr : REAL;
	sin_out : REAL;
	phi : REAL;
	frequency : REAL;
	MC_BR_CyclicWrite_0 : MC_BR_CyclicWrite;
	MC_BR_WriteParID_0 : MC_BR_WriteParID;
	initParIDs : BOOL;
	MC_BR_WriteParID_1 : MC_BR_WriteParID;
END_VAR
```

#### Main.st
```iecst
PROGRAM _INIT

	MaxCurr := 1.5;		 // Max current [A]
	frequency := 49.0;	 // frequency [Hz]

	initParIDs := TRUE;

END_PROGRAM

PROGRAM _CYCLIC

	MC_Power_0.Enable := Run;
	MC_Power_0.Axis := ADR(gAxisVibC);
	MC_Power_0();

	IF MC_Power_0.Status THEN
//		............................ Wave Generator ..................................
//		...............o......o.......................................................
//		............o............o....................................................
//		..........o................o..................................................
//		........o....................o................................................
//		.......o......................o...............................................
//		.....o..........................o.............................................
//		....o............................o............................................
//		...o...............................o..........................................
//		....................................o..............................o..........
//		.....................................o............................o...........
//		......................................o..........................o............
//		........................................o......................o..............
//		.........................................o....................o...............
//		...........................................o................o.................
//		.............................................o............o...................
//		................................................o......o......................

		amplitude_out := LIMIT(-MaxCurr,amplitude_out,MaxCurr);
		sin_out := amplitude_out*SIN(phi);
		phi := fmod(phi + frequency*2*PI*CYCLE_TIME_s, 2*PI);
	ELSE
		sin_out := 0.0;
	END_IF

	// Write sine wave to vibrator parID (Will be interpolated in drive with SPT Function Block)
	MC_BR_CyclicWrite_0.Enable := Run;
	MC_BR_CyclicWrite_0.Axis := ADR(gAxisVibC);
	MC_BR_CyclicWrite_0.DataType := ncPAR_TYP_REAL;
	MC_BR_CyclicWrite_0.DataAddress := ADR(sin_out);
	MC_BR_CyclicWrite_0.ParID := ACP10PAR_USER_R4_VAR1;
	MC_BR_CyclicWrite_0();

	IF initParIDs THEN

		// Have to overwrite in code to "cheat" the drive into using Current Controller for 1 phase control (doesn't work in parameter table)
		MC_BR_WriteParID_0.Execute 			:= TRUE;
		MC_BR_WriteParID_0.Axis 			:= ADR(gAxisVibC);
		MC_BR_WriteParID_0.ParID 			:= ACP10PAR_CONTROLLER_MODE;
		MC_BR_WriteParID_0.DataType 		:= ncPAR_TYP_USINT;
		MC_BR_WriteParID_0.DataAddress	 	:= ADR(CONTROLLER_MODE_CURR_CTRL); // 5=Current Controller
		MC_BR_WriteParID_0();

		MC_BR_WriteParID_1.Execute 			:= TRUE;
		MC_BR_WriteParID_1.Axis 			:= ADR(gAxisVibC);
		MC_BR_WriteParID_1.ParID 			:= ACP10PAR_ICTRL_SET_PARID;	// SetPoint to ACP10 Current Controller
		MC_BR_WriteParID_1.DataType 		:= ncPAR_TYP_UINT;
		MC_BR_WriteParID_1.DataAddress 		:= ADR(PARID_IPL1_OUT);
		MC_BR_WriteParID_1();

		IF MC_BR_WriteParID_0.Done AND MC_BR_WriteParID_1.Done THEN
			MC_BR_WriteParID_0.Execute := FALSE;
			MC_BR_WriteParID_0();
			MC_BR_WriteParID_1.Execute := FALSE;
			MC_BR_WriteParID_1();

			initParIDs := FALSE; // Done
		END_IF

	END_IF

END_PROGRAM

PROGRAM _EXIT

END_PROGRAM
```

Listed in the project but not available here: Logical/Libraries/brdkMU/brdkMU.typ, Logical/Libraries/brdkMU/brdkUM.typ, Logical/Libraries/brdkMU/brdkMU.var, Logical/Libraries/brdkMU/brdkMU.fun, Logical/Libraries/brdkMU/brdkEMStateToA.c, Logical/Libraries/brdkMU/brdkEM_func.h, Logical/Libraries/brdkMU/brdkCMChangeParent.c, Logical/Libraries/brdkMU/brdkCM_func.h, Logical/Libraries/brdkMU/brdkUM.c, Logical/Libraries/brdkMU/brdkUM_func.h, Logical/Libraries/brdkMU/brdkUM_func.c, Logical/Libraries/brdkMU/brdkMU_func.h, Logical/Libraries/brdkMU/brdkMU_func.c, Logical/Libraries/brdkSIM/Constants.var, Logical/Libraries/brdkSIM/brdkSIM.fun, Logical/Libraries/brdkCSV/Types.typ, Logical/Libraries/brdkCSV/Constants.var, Logical/Libraries/brdkPV/brdkPV.typ, Logical/Libraries/legoCM20/legocm20.var, Logical/Libraries/brdkFile/brdkFileCreateSubFolders.c, Logical/Libraries/brdkFile/brdkFile_func.h, Logical/Libraries/brdkFile/brdkFile_func.c, Logical/Libraries/brdkJSON/brdkJSON.var, Logical/Libraries/brdkSTR/brdkSTR.typ, Logical/Libraries/brdkSTR/brdkSTR.var, Logical/Libraries/brdkSTR/brdkStrAToDint.c, Logical/Libraries/brdkSTR/brdkStrAToDTStructure.c, Logical/Libraries/brdkSTR/brdkStrAToUdint.c, Logical/Libraries/brdkSTR/brdkStrCat.c, Logical/Libraries/brdkSTR/brdkStrCatAtChar.c, Logical/Libraries/brdkSTR/brdkStrCharAt.c, Logical/Libraries/brdkSTR/brdkStrCharCount.c, Logical/Libraries/brdkSTR/brdkStrCmp.c, Logical/Libraries/brdkSTR/brdkStrCpy.c, Logical/Libraries/brdkSTR/brdkStrCrc32.c, Logical/Libraries/brdkSTR/brdkStrDintToA.c, Logical/Libraries/brdkSTR/brdkStrEncode.c, Logical/Libraries/brdkSTR/brdkStrFill.c, Logical/Libraries/brdkSTR/brdkStrFillUp.c, Logical/Libraries/brdkSTR/brdkStrIndexOf.c, Logical/Libraries/brdkSTR/brdkStrInsertAtPos.c, Logical/Libraries/brdkSTR/brdkStrIsEmpty.c, Logical/Libraries/brdkSTR/brdkStrJoin.c, Logical/Libraries/brdkSTR/brdkStrLen.c, Logical/Libraries/brdkSTR/brdkStrMemClear.c, Logical/Libraries/brdkSTR/brdkStrMemCmp.c, Logical/Libraries/brdkSTR/brdkStrMemCpy.c, Logical/Libraries/brdkSTR/brdkStrMemMove.c, Logical/Libraries/brdkSTR/brdkStrMemSet.c, Logical/Libraries/brdkSTR/brdkStrMove.c, Logical/Libraries/brdkSTR/brdkStrNAToDint.c, Logical/Libraries/brdkSTR/brdkStrNCpy.c, Logical/Libraries/brdkSTR/brdkStrRemove.c, Logical/Libraries/brdkSTR/brdkStrRepeat.c, Logical/Libraries/brdkSTR/brdkStrReplace.c, Logical/Libraries/brdkSTR/brdkStrReverse.c, Logical/Libraries/brdkSTR/brdkStrReverseWords.c, Logical/Libraries/brdkSTR/brdkStrSearch.c, Logical/Libraries/brdkSTR/brdkStrSlice.c, Logical/Libraries/brdkSTR/brdkStrSplit.c, Logical/Libraries/brdkSTR/brdkStrSubDintSearch.c, Logical/Libraries/brdkSTR/brdkStrSubStr.c, Logical/Libraries/brdkSTR/brdkStrSubStrSearch.c, Logical/Libraries/brdkSTR/brdkStrToDec.c, Logical/Libraries/brdkSTR/brdkStrToHex.c, Logical/Libraries/brdkSTR/brdkStrToLowerCase.c, Logical/Libraries/brdkSTR/brdkStrToUpperCase.c, Logical/Libraries/brdkSTR/brdkStrToUpperCaseWords.c, Logical/Libraries/brdkSTR/brdkStrTrim.c, Logical/Libraries/brdkSTR/brdkStrWord.c, Logical/Libraries/Goertzel/freqHelp.typ, Logical/services/machine/updateEWU/local.typ, Logical/services/alarm/alarm/local.typ, Logical/services/file/file/local.typ, Logical/services/recipe/recipe/types.typ, Logical/acp10etxen
